// TIA Portal V17 program export: 0 tag tables, 0 data types, 40 data blocks, 87 code blocks (in call order from the OBs), 109 instance data blocks

DATA_BLOCK "General_DB"   // DB47
{ S7_Optimized_Access := 'TRUE' }
VERSION : 0.1
// stored: AutoNumber false, DBAccessibleFromOPCUA true, DBAccessibleFromWebserver true, IsOnlyStoredInLoadMemory false, IsRetainMemResEnabled false, IsWriteProtectedInAS false, MemoryReserve 100
   VAR
      Initial : Bool;
      "Reset HMI Prep" : Bool;
      "Reset HMI ST" : Bool;
      "Reset HMI Blend" : Bool;
      "Reset Scada" : Bool;
      Reset : Bool;
      Reset_Dose : Bool;
      Sim_Mode : Bool;   // 1 Simulation
      Sim_ON : Bool;
      Sim_OFF : Bool;
      Man_Initi : Bool;
      LDT_PLC : Date_And_Time;
      LDT_retval : Int;
      CIP_Line1_Open : Struct
         "CIP Tank_T01" : Bool;
         "CIP Line_T01" : Bool;
         "CIP Tank_T02" : Bool;
         "CIP Line_T02" : Bool;
         "CIP Tank_T03" : Bool;
         "CIP Line_T03" : Bool;
         "CIP Tank_T04" : Bool;
         "CIP Line_T04" : Bool;
         "CIP Tank_T05" : Bool;
         "CIP Line_T05" : Bool;
         "CIP Tank_T06" : Bool;
         "CIP Line_T06" : Bool;
         "CIP Tank_T07" : Bool;
         "CIP Line_T07" : Bool;
         "CIP Tank_T08" : Bool;
         "CIP Line_T08" : Bool;
         "CIP Tank_T09" : Bool;
         "CIP Line_T09" : Bool;
         "CIP Tank_T10" : Bool;
         "CIP Line_T10" : Bool;
         "CIP Tank_T11" : Bool;
         "CIP Line_T11" : Bool;
         "CIP Tank_T12" : Bool;
         "CIP Line_T12" : Bool;
         "CIP Tank_T13" : Bool;
         "CIP Line_T13" : Bool;
         CIP_Tank : Bool;
         CIP_Line : Bool;
      END_STRUCT;
      CIP_Line2_Open : Struct
         "CIP Tank_T1" : Bool;
         "CIP Line_T1" : Bool;
         "CIP Tank_T2" : Bool;
         "CIP Line_T2" : Bool;
         "CIP Tank_T3" : Bool;
         "CIP Line_T3" : Bool;
         "CIP Tank_T4" : Bool;
         "CIP Line_T4" : Bool;
         "CIP Tank_T5" : Bool;
         "CIP Line_T5" : Bool;
         "CIP Tank_T6" : Bool;
         "CIP Line_T6" : Bool;
         "CIP Tank_T7" : Bool;
         "CIP Line_T7" : Bool;
         "CIP Tank_T8" : Bool;
         "CIP Line_T8" : Bool;
         "CIP Tank_T9" : Bool;
         "CIP Line_T9" : Bool;
         "CIP Tank_T10" : Bool;
         "CIP Line_T10" : Bool;
         CIP_Tank : Bool;
         CIP_Line : Bool;
      END_STRUCT;
      "Bypass CIP Signal Storage" : Bool;
      "Bypass CIP Signal Homomixer" : Bool;
      "Testing FB Valve" : Struct
         Preparation : Bool;
         Homomixer : Bool;
         Blending : Bool;
         Storage : Bool;
      END_STRUCT;
      "Testing FB Motor" : Struct
         "MCC Blending" : Bool;
         "MCC Preparation" : Bool;
      END_STRUCT;
      "CIP Drain Time" : Struct
         BlendingCluster1 : TOF_TIME;
         BlendingCluster2 : TOF_TIME;
         "Preparation_02.20" : TOF_TIME;
         "Preparation_05.20" : TOF_TIME;
         Homomixer : TOF_TIME;
         "Storage_29.06" : TOF_TIME;
         "Storage_39.06" : TOF_TIME;
         HMI_Input : Struct
            BlendingCluster1 : Int := 60;
            BlendingCluster2 : Int := 60;
            "Preparation_02.20" : Int := 60;
            "Preparation_05.20" : Int := 60;
            Homomixer : Int := 60;
            "Storage_29.06" : Int := 60;
            "Storage_39.06" : Int := 60;
         END_STRUCT;
         Actual : Struct
            BlendingCluster1 : DInt;
            BlendingCluster2 : DInt;
            "Preparation_02.20" : DInt;
            "Preparation_05.20" : DInt;
            Homomixer : DInt;
            "Storage_29.06" : DInt;
            "Storage_39.06" : DInt;
         END_STRUCT;
      END_STRUCT;
   END_VAR
BEGIN
   "CIP Drain Time".BlendingCluster1.PT := T#1m;
   "CIP Drain Time".BlendingCluster2.PT := T#1m;
   "CIP Drain Time"."Preparation_02.20".PT := T#1m;
   "CIP Drain Time"."Preparation_05.20".PT := T#1m;
   "CIP Drain Time".Homomixer.PT := T#1m;
   "CIP Drain Time"."Storage_29.06".PT := T#1m;
   "CIP Drain Time"."Storage_39.06".PT := T#1m;
END_DATA_BLOCK

DATA_BLOCK "General_Blend"   // DB33
{ S7_Optimized_Access := 'TRUE' }
VERSION : 0.1
// stored: AutoNumber true, DBAccessibleFromOPCUA true, DBAccessibleFromWebserver true, IsOnlyStoredInLoadMemory false, IsRetainMemResEnabled false, IsWriteProtectedInAS false, MemoryReserve 100
   VAR
      Drain_ON_OFF_THE1 : Bool;
      Drain_ON_OFF_THE2 : Bool;
      Blend_Cluster1 : Struct
         CIP_Line1 : Struct
            "CIP Enable" : Bool;
            "CIP Request" : Bool;
            V_Cmd : Bool;
            P_Cmd : Bool;
            P_SP : Real;
         END_STRUCT;
         CIP_Line2 : Struct
            "CIP Enable" : Bool;
            "CIP Request" : Bool;
            V_Cmd : Bool;
            P_Cmd : Bool;
            P_SP : Real;
         END_STRUCT;
         CIP_Line3 : Struct
            "CIP Enable" : Bool;
            "CIP Request" : Bool;
            V_Cmd : Bool;
            P_Cmd : Bool;
            P_SP : Real;
         END_STRUCT;
         ptrig : Bool;
      END_STRUCT;
      Blend_Cluster2 : Struct
         CIP_Line1 : Struct
            "CIP Enable" : Bool;
            "CIP Request" : Bool;
            V_Cmd : Bool;
            P_Cmd : Bool;
            P_SP : Real;
         END_STRUCT;
         CIP_Line2 : Struct
            "CIP Enable" : Bool;
            "CIP Request" : Bool;
            V_Cmd : Bool;
            P_Cmd : Bool;
            P_SP : Real;
         END_STRUCT;
         CIP_Line3 : Struct
            "CIP Enable" : Bool;
            "CIP Request" : Bool;
            V_Cmd : Bool;
            P_Cmd : Bool;
            P_SP : Real;
         END_STRUCT;
         ptrig : Bool;
      END_STRUCT;
      CIP_Bypass : Bool;
      "THE-4" : Struct
         "Timer" : TON_TIME;
         MSec { S7_SetPoint := 'True'} : DInt;
         Sec : DInt := 10;
         Act : DInt;
      END_STRUCT;
      "THE-5" : Struct
         "Timer" : TON_TIME;
         MSec { S7_SetPoint := 'True'} : DInt;
         Sec : DInt := 10;
         Act : DInt;
      END_STRUCT;
      Sugar : Struct
         "In Process" : Struct
            "T-20" : Bool;
            "T-21" : Bool;
            "T-30" : Bool;
            "T-31" : Bool;
            "T-40" : Bool;
            "T-41" : Bool;
         END_STRUCT;
      END_STRUCT;
   END_VAR
BEGIN
END_DATA_BLOCK

DATA_BLOCK "Gen_Storage"   // DB15
{ S7_Optimized_Access := 'TRUE' }
VERSION : 0.1
// stored: AutoNumber false, DBAccessibleFromOPCUA true, DBAccessibleFromWebserver true, IsOnlyStoredInLoadMemory false, IsRetainMemResEnabled false, IsWriteProtectedInAS false, MemoryReserve 100
   VAR
      "Timer" : Struct
         Off_DrainIn_23 : TOF_TIME;
         Off_DrainIn_24_1 { S7_SetPoint := 'True'} : TOF_TIME;
         Off_DrainIn_24_2 { S7_SetPoint := 'True'} : TOF_TIME;
         Off_DrainIn_33 { S7_SetPoint := 'True'} : TOF_TIME;
         Off_DrainIn_34 { S7_SetPoint := 'True'} : TOF_TIME;
         Off_DrainIn_35 { S7_SetPoint := 'True'} : TOF_TIME;
         Off_DrainIn_79_1 { S7_SetPoint := 'True'} : TOF_TIME;
         Off_DrainIn_79_2 { S7_SetPoint := 'True'} : TOF_TIME;
         Off_DrainIn_79_3 { S7_SetPoint := 'True'} : TOF_TIME;
         Off_DrainIn_81 { S7_SetPoint := 'True'} : TOF_TIME;
         Off_DrainIn_84 { S7_SetPoint := 'True'} : TOF_TIME;
         Off_DrainIn_85 { S7_SetPoint := 'True'} : TOF_TIME;
      END_STRUCT;
      "THE4 CIP" : Struct
         "CIP Enable" : Bool;
         "CIP Request" : Bool;
         "CIP Line OK" : Bool;
         "CIP on Prog" : Bool;
         V_CIP_Cmd : Bool;
         p_trig : Bool;
      END_STRUCT;
      "THE5 CIP" : Struct
         "CIP Enable" : Bool;
         "CIP Request" : Bool;
         "CIP Line OK" : Bool;
         "CIP on Prog" : Bool;
         V_CIP_Cmd : Bool;
         p_trig : Bool;
      END_STRUCT;
   END_VAR
BEGIN
   "Timer".Off_DrainIn_23.PT := T#3s;
   "Timer".Off_DrainIn_24_1.PT := T#3s;
   "Timer".Off_DrainIn_33.PT := T#3s;
   "Timer".Off_DrainIn_34.PT := T#3s;
   "Timer".Off_DrainIn_35.PT := T#3s;
   "Timer".Off_DrainIn_79_1.PT := T#3s;
   "Timer".Off_DrainIn_81.PT := T#3s;
   "Timer".Off_DrainIn_84.PT := T#3s;
   "Timer".Off_DrainIn_85.PT := T#3s;
END_DATA_BLOCK

DATA_BLOCK "General Preparation"   // DB59
{ S7_Optimized_Access := 'TRUE' }
VERSION : 0.1
// stored: AutoNumber true, DBAccessibleFromOPCUA true, DBAccessibleFromWebserver true, IsOnlyStoredInLoadMemory false, IsRetainMemResEnabled false, IsWriteProtectedInAS false, MemoryReserve 100
   VAR
      "Header 1" : Struct
         "CIP Enable" : Bool;
         "CIP Request" : Bool;
         "CIP Line OK" : Bool;
         "CIP on Prog" : Bool;
         V_CIP_Cmd : Bool;
         p_trig : Bool;
      END_STRUCT;
      "Header 2" : Struct
         "CIP Enable" : Bool;
         "CIP Request" : Bool;
         "CIP Line OK" : Bool;
         "CIP on Prog" : Bool;
         V_CIP_Cmd : Bool;
         p_trig : Bool;
      END_STRUCT;
      "Blend OSA" : Struct
         "CIP Enable_T-06 Cmd" : Bool;
         "CIP Enable_T-07 Cmd" : Bool;
         "CIP Enable_T-08 Cmd" : Bool;
         "CIP Request" : Bool;
         "CIP on Prog" : Bool;
         "CIP EN T-06" : Bool;
         "CIP EN T-07" : Bool;
         "CIP EN T-08" : Bool;
      END_STRUCT;
      "Tipper 1" : Struct
         "CIP Enable Cmd" : Bool;
         "CIP Request" : Bool;
         "CIP on Prog" : Bool;
         "CIP EN" : Bool;
      END_STRUCT;
      "Tipper 2" : Struct
         "CIP Enable_T-03 Cmd" : Bool;
         "CIP Enable_T-04 Cmd" : Bool;
         "CIP Request" : Bool;
         "CIP on Prog" : Bool;
         "CIP EN T-03" : Bool;
         "CIP EN T-04" : Bool;
      END_STRUCT;
      CIP_Bypass : Bool;
      Reset_Totalizer : Struct
         "FT_T-51" : Bool;
         "FT_T-02" : Bool;
         "FT_T-3" : Bool;
         "FT_T-4" : Bool;
         "FT_T-5" : Bool;
         "FT_T-6" : Bool;
         "FT_T-7" : Bool;
         "FT_T-8" : Bool;
         "FT_T-9" : Bool;
         "FT_T-10" : Bool;
      END_STRUCT;
      CV_Value_Manual : Real;
   END_VAR
   VAR RETAIN
      Tank_Name : Struct
         ChiliAwetan1 : String := 'Chili Awetan 1';
         ChiliAwetan2 : String := 'Chili Awetan 2';
         ChiliAwetan3 : String := 'Chili Awetan 3';
         Tomato : String := 'Tomato';
         ChiliFresh1 : String := 'Chili Fresh 1';
         ChiliFresh2 : String := 'Chili Fresh 2';
         ChiliFresh3 : String := 'Chili Fresh 3';
         Garlic : String := 'Garlic';
         Vinegar : String := 'Vinegar';
         HotWater : String := 'Hot Water';
         free11 : String;
      END_STRUCT;
   END_VAR
BEGIN
END_DATA_BLOCK

DATA_BLOCK "General Buffer"   // DB63
{ S7_Optimized_Access := 'TRUE' }
VERSION : 0.1
// stored: AutoNumber true, DBAccessibleFromOPCUA true, DBAccessibleFromWebserver true, IsOnlyStoredInLoadMemory false, IsRetainMemResEnabled false, IsWriteProtectedInAS false, MemoryReserve 100
   VAR
      "CIP Enable" : Struct
         Cluster1_Line3 : Bool;
         Cluster2_Line1 : Bool;
         Cluster2_Line2 : Bool;
         Cluster2_Line3 : Bool;
      END_STRUCT;
      "CIP Line Open" : Struct
         Cluster1_Line3 : Bool;
         Cluster2_Line1 : Bool;
         Cluster2_Line2 : Bool;
         Cluster2_Line3 : Bool;
      END_STRUCT;
   END_VAR
BEGIN
END_DATA_BLOCK

DATA_BLOCK "CIP_CIP_to_Sto"   // DB190
{ S7_Optimized_Access := 'FALSE' }
VERSION : 0.1
// stored: AutoNumber false, DBAccessibleFromOPCUA true, DBAccessibleFromWebserver true, IsOnlyStoredInLoadMemory false, IsWriteProtectedInAS false
   VAR
      HeatBeat : Bool;
      CIP_Ready : Bool;   // Cip Kitchen Ready
      CIP_Inprogress : Bool;   // Reqquest approved
      CIP_Complete : Bool;
      Valve_Line_Return_Open : Bool;
      Spare : Bool;
      Spare_1 : Bool;
      Spare_2 : Bool;
      Spare_3 : Bool;
      Spare_4 : Bool;
      Spare_5 : Bool;
      Spare_6 : Bool;
      Spare_7 : Bool;
      Spare_8 : Bool;
      Spare_9 : Bool;
      Spare_10 : Bool;
      Data_Real : Real;
      Data_Real_1 : Real;
      Data_Real_2 : Real;
      Data_Real_3 : Real;
      Data_Real_4 : Real;
      Data_Real_5 : Real;
      Data_Real_6 : Real;
      Data_Real_7 : Real;
   END_VAR
BEGIN
END_DATA_BLOCK

DATA_BLOCK "CIP_Sto_to_CIP"   // DB191
{ S7_Optimized_Access := 'FALSE' }
VERSION : 0.1
// stored: AutoNumber false, DBAccessibleFromOPCUA true, DBAccessibleFromWebserver true, IsOnlyStoredInLoadMemory false, IsWriteProtectedInAS false
   VAR
      HeatBeat : Bool;
      CIP_Request : Bool;   // Cip Kitchen Ready
      ReturnPump_ON : Bool;   // Reqquest approved
      CIP_Complete : Bool;
      Valve_Line_Supply_Open : Bool;
      Spare : Bool;
      Spare_1 : Bool;
      Spare_2 : Bool;
      Spare_3 : Bool;
      Spare_4 : Bool;
      Spare_5 : Bool;
      Spare_6 : Bool;
      Spare_7 : Bool;
      Spare_8 : Bool;
      Spare_9 : Bool;
      Spare_10 : Bool;
      Data_Real : Real;
      Data_Real_1 : Real;
      Data_Real_2 : Real;
      Data_Real_3 : Real;
      Data_Real_4 : Real;
      Data_Real_5 : Real;
      Data_Real_6 : Real;
      Data_Real_7 : Real;
   END_VAR
BEGIN
END_DATA_BLOCK

DATA_BLOCK "CommSett_DB"   // DB10
{ S7_Optimized_Access := 'TRUE' }
VERSION : 0.1
// stored: AutoNumber false, DBAccessibleFromOPCUA true, DBAccessibleFromWebserver true, IsOnlyStoredInLoadMemory false, IsRetainMemResEnabled false, IsWriteProtectedInAS false, MemoryReserve 100
   VAR
      THE1_put : "typePut";
      THE1_get { S7_SetPoint := 'True'} : "typeGet";
      THE1_diagnostic { S7_SetPoint := 'True'} : "typeDiagnostic";
      THE2_put : "typePut";
      THE2_get { S7_SetPoint := 'True'} : "typeGet";
      THE2_diagnostic { S7_SetPoint := 'True'} : "typeDiagnostic";
      THE1_Comm_Error { S7_SetPoint := 'True'} : Bool;
      THE2_Comm_Error : Bool;
      THE1_Comm : Array[0..10] of Byte;
      THE2_Comm : Array[0..10] of Byte;
      CIP_put : "typePut";
      CIP_get { S7_SetPoint := 'True'} : "typeGet";
      CIP_diagnostic { S7_SetPoint := 'True'} : "typeDiagnostic";
      CIP_Comm_Error { S7_SetPoint := 'True'} : Bool;
      CIP_Comm : Array[0..10] of Byte;
   END_VAR
BEGIN
   THE1_put.connectionId := 16#100;
   THE1_get.connectionId := 16#100;
   THE2_put.connectionId := 16#101;
   THE2_get.connectionId := 16#101;
   CIP_put.connectionId := 16#102;
   CIP_get.connectionId := 16#102;
END_DATA_BLOCK

DATA_BLOCK "Data_block_1"   // DB196
{ S7_Optimized_Access := 'FALSE'; DB_Accessible_From_OPC_UA := 'FALSE' }
VERSION : 0.1
// stored: AutoNumber false, DBAccessibleFromOPCUA false, DBAccessibleFromWebserver false, IsOnlyStoredInLoadMemory false, IsWriteProtectedInAS false
   VAR
      FromTHE4 : Array[0..50] of Byte;
   END_VAR
BEGIN
END_DATA_BLOCK

DATA_BLOCK "THE1_From_BT_To_Mixing"   // DB194
{ S7_Optimized_Access := 'FALSE' }
VERSION : 0.1
// stored: AutoNumber false, DBAccessibleFromOPCUA true, DBAccessibleFromWebserver true, IsOnlyStoredInLoadMemory false, IsWriteProtectedInAS false
   VAR RETAIN
      HeartBeat : Bool := TRUE;
      CIPEnable : Bool;
      LineProd_Open : Bool;
      LineCIP_Open : Bool;
      _free_4 : Bool;
      _free_5 : Bool;
      _free_6 : Bool;
      _free_7 : Bool;
      ProductRequest : Bool;
      _free_09 : Bool;
      _free_10 : Bool;
      _free_11 : Bool;
      _free_12 : Bool;
      _free_13 : Bool;
      _free_14 : Bool;
      _free_15 : Bool;
      _free_real2 : Real;
      _free_real6 : Real := 20000.0;
      _free_real10 : Real;
      _free_real14 : Real;
      _free_real18 : Real;
      _free_real22 : Real;
      _free_real26 : Real;
      _free_real30 : Real;
      FromTHE1Byte1 : Byte;
      FromTHE1Byte2 : Byte;
      FromTHE1Byte3 : Byte;
      FromTHE1Byte4 : Byte;
   END_VAR
BEGIN
END_DATA_BLOCK

DATA_BLOCK "THE1_From_Mixing_To_BT"   // DB195
{ S7_Optimized_Access := 'FALSE' }
VERSION : 0.1
// stored: AutoNumber false, DBAccessibleFromOPCUA true, DBAccessibleFromWebserver true, IsOnlyStoredInLoadMemory false, IsWriteProtectedInAS false
   VAR RETAIN
      HeartBeat : Bool;
      CIPRequest : Bool;
      MixProofFlip : Bool;
      Drain_valve : Bool;
      _free_4 : Bool;
      _free_5 : Bool;
      _free_6 : Bool;
      _free_7 : Bool;
      ProductAvailable : Bool;
      ProductTransferInProgress : Bool;
      _free_10 : Bool;
      _free_11 : Bool;
      _free_12 : Bool;
      _free_13 : Bool;
      _free_14 : Bool;
      _free_15 : Bool;
      _free_real2 : Real := 52.25618;
      _free_real6 : Real := 93.70135;
      _free_real10 : Real := 95.52147;
      _free_real14 : Real := 90.2006;
      _free_real18 : Real;
      _free_real22 : Real;
      _free_real26 : Real;
      _free_real30 : Real;
      ForTHE1_Byte1 : Byte;
      ForTHE1_Byte2 : Byte;
      ForTHE1_Byte3 : Byte;
      ForTHE1_Byte4 : Byte;
   END_VAR
BEGIN
END_DATA_BLOCK

DATA_BLOCK "THE2_From_BT_To_Mixing"   // DB198
{ S7_Optimized_Access := 'FALSE' }
VERSION : 0.1
// stored: AutoNumber false, DBAccessibleFromOPCUA true, DBAccessibleFromWebserver true, IsOnlyStoredInLoadMemory false, IsWriteProtectedInAS false
   VAR RETAIN
      HeartBeat : Bool := TRUE;
      CIPEnable : Bool;
      LineProd_Open : Bool;
      LineCIP_Open : Bool;
      _free_4 : Bool;
      _free_5 : Bool;
      _free_6 : Bool;
      _free_7 : Bool;
      ProductRequest : Bool;
      _free_09 : Bool;
      _free_10 : Bool;
      _free_11 : Bool;
      _free_12 : Bool;
      _free_13 : Bool;
      _free_14 : Bool;
      _free_15 : Bool;
      _free_real2 : Real;
      _free_real6 : Real := 20000.0;
      _free_real10 : Real;
      _free_real14 : Real;
      _free_real18 : Real;
      _free_real22 : Real;
      _free_real26 : Real;
      _free_real30 : Real;
      FromTHE2Byte1 : Byte;
      FromTHE2Byte2 : Byte;
      FromTHE2Byte3 : Byte;
      FromTHE2Byte4 : Byte;
   END_VAR
BEGIN
END_DATA_BLOCK

DATA_BLOCK "THE2_From_Mixing_To_BT"   // DB199
{ S7_Optimized_Access := 'FALSE' }
VERSION : 0.1
// stored: AutoNumber false, DBAccessibleFromOPCUA true, DBAccessibleFromWebserver true, IsOnlyStoredInLoadMemory false, IsWriteProtectedInAS false
   VAR RETAIN
      HeartBeat : Bool;
      CIPRequest : Bool;
      MixProofFlip : Bool;
      Drain_valve : Bool;
      _free_4 : Bool;
      _free_5 : Bool;
      _free_6 : Bool;
      _free_7 : Bool;
      ProductAvailable : Bool;
      ProductTransferInProgress : Bool;
      _free_10 : Bool;
      _free_11 : Bool;
      _free_12 : Bool;
      _free_13 : Bool;
      _free_14 : Bool;
      _free_15 : Bool;
      _free_real2 : Real := 52.25618;
      _free_real6 : Real := 93.70135;
      _free_real10 : Real := 95.52147;
      _free_real14 : Real := 90.2006;
      _free_real18 : Real;
      _free_real22 : Real;
      _free_real26 : Real;
      _free_real30 : Real;
      ForTHE2_Byte1 : Byte;
      ForTHE2_Byte2 : Byte;
      ForTHE2_Byte3 : Byte;
      ForTHE2_Byte4 : Byte;
   END_VAR
BEGIN
END_DATA_BLOCK

DATA_BLOCK "MB to Osa"   // DB265
{ S7_Optimized_Access := 'FALSE' }
VERSION : 0.1
// stored: AutoNumber false, DBAccessibleFromOPCUA true, DBAccessibleFromWebserver true, IsOnlyStoredInLoadMemory false, IsWriteProtectedInAS false
   VAR
      HeartBeat : Bool;   // Clock 1Hz
      ChiliFresh1_Prod_Req : Bool;
      ChiliFresh2_Prod_Req : Bool;
      ChiliFresh3_Prod_Req : Bool;
      ChiliFresh1_Line_OK : Bool;
      ChiliFresh2_Line_OK : Bool;
      ChiliFresh3_Line_OK : Bool;
      ChiliFresh1_CIP_Enable : Bool;
      ChiliFresh2_CIP_Enable : Bool;
      ChiliFresh3_CIP_Enable : Bool;
      freeBool11 : Bool;
      freeBool12 : Bool;
      freeBool13 : Bool;
      freeBool14 : Bool;
      freeBool15 : Bool;
      freeBool16 : Bool;
      freeBool17 : Bool;
   END_VAR
BEGIN
END_DATA_BLOCK

DATA_BLOCK "Osa to MB"   // DB264
{ S7_Optimized_Access := 'FALSE' }
VERSION : 0.1
// stored: AutoNumber false, DBAccessibleFromOPCUA true, DBAccessibleFromWebserver true, IsOnlyStoredInLoadMemory false, IsWriteProtectedInAS false
   VAR
      HeartBeat : Bool;   // Clock 1hz
      Product_Ready : Bool;
      Product_LineOpen : Bool;
      Product_SupplyON : Bool;
      Product_Transfer_Complete : Bool;
      freeBool5 : Bool;
      freeBool6 : Bool;
      freeBool7 : Bool;
      freeBool8 : Bool;
      freeBool9 : Bool;
      freeBool10 : Bool;
      freeBool11 : Bool;
      freeBool12 : Bool;
      freeBool13 : Bool;
      freeBool14 : Bool;
      freeBool15 : Bool;
      freeBool16 : Bool;
      freeBool17 : Bool;
      freeBool18 : Bool;
      freeBool19 : Bool;
      freeBool20 : Bool;
      freeBool21 : Bool;
      freeBool22 : Bool;
      freeBool23 : Bool;
   END_VAR
BEGIN
END_DATA_BLOCK

DATA_BLOCK "CIP_to_Mix"   // DB220
{ S7_Optimized_Access := 'FALSE' }
VERSION : 0.1
// stored: AutoNumber false, DBAccessibleFromOPCUA true, DBAccessibleFromWebserver true, IsOnlyStoredInLoadMemory false, IsWriteProtectedInAS false
   VAR
      HeartBeat : Bool := TRUE;
      CIP_RequestOK : Struct
         Header : Struct
            Header_CIP_RequestOK : Bool;
         END_STRUCT;
         "Chili Awetan" : Struct
            "T-02.00_CIP_RequestOK" : Bool;
            "T-03.00_CIP_RequestOK" : Bool;
            "T-04.00_CIP_RequestOK" : Bool;
         END_STRUCT;
         Tomato : Struct
            "T-05.00_CIP_RequestOK" : Bool;
         END_STRUCT;
         ChiliFresh : Struct
            "T-06.00_CIP_RequestOK" : Bool;
            "T-07.00_CIP_RequestOK" : Bool;
            "T-08.00_CIP_RequestOK" : Bool;
         END_STRUCT;
         Garlic : Struct
            "T-09.00_CIP_RequestOK" : Bool;
         END_STRUCT;
         Vinegar : Struct
            "T-10.00_CIP_RequestOK" : Bool;
         END_STRUCT;
         Homomixer : Struct
            "T-12.00_CIP_RequestOK" : Bool;
            "T-13.00_CIP_RequestOK" : Bool;
            "T-14.00_CIP_RequestOK" : Bool;
         END_STRUCT;
         "Blending Cluster 1" : Struct
            "T-20.00_CIP_RequestOK" : Bool;
            "T-21.00_CIP_RequestOK" : Bool;
            "T-30.00_CIP_RequestOK" : Bool;
            Blending_Cluster1_LineProduct_RequestOK : Bool;
            Free_CIP_RequestOK_1 : Bool;
            Free_CIP_RequestOK_2 : Bool;
         END_STRUCT;
         "Blending Cluster 2" : Struct
            "T-31.00_CIP_RequestOK" : Bool;
            "T-40.00_CIP_RequestOK" : Bool;
            "T-41.00_CIP_RequestOK" : Bool;
            Blending_Cluster2_LineProduct_RequestOK : Bool;
            Free_CIP_RequestOK_1 : Bool;
            Free_CIP_RequestOK_2 : Bool;
         END_STRUCT;
         "Rework Cluster 1" : Struct
            "T-22.00_CIP_RequestOK" : Bool;
         END_STRUCT;
         "Rework Cluster 2" : Struct
            "T-32.00_CIP_RequestOK" : Bool;
         END_STRUCT;
         "Buffer Cluster 1" : Struct
            "T-61.00_CIP_RequestOK" : Bool;
            "T-62.00_CIP_RequestOK" : Bool;
            "T61&T62_CIP_LineToPasteur_RequestOK" : Bool;
            "T-63.00_CIP_RequestOK" : Bool;
            "T-64.00_CIP_RequestOK" : Bool;
            "T63&T64_CIP_LineToPasteur_RequestOK" : Bool;
         END_STRUCT;
         "Buffer Cluster 2" : Struct
            "T-65.00_CIP_RequestOK" : Bool;
            "T-66.00_CIP_RequestOK" : Bool;
            "T65&T66_CIP_LineToPasteur_RequestOK" : Bool;
            "T-67.00_CIP_RequestOK" : Bool;
            "T-68.00_CIP_RequestOK" : Bool;
            "T67&T68_CIP_LineToPasteur_RequestOK" : Bool;
         END_STRUCT;
         "Storage THE 4" : Struct
            "T-23.00_CIP_RequestOK" : Bool;
            "T-24.00_CIP_RequestOK" : Bool;
            THE4_LineProduct_CIP_RequestOK : Bool;
         END_STRUCT;
         "Storage THE 5" : Struct
            "T-33.00_CIP_Tank_RequestOK" : Bool;
            "T-34.00_CIP_Tank_RequestOK" : Bool;
            "T33&T34_CIP_Line_RequestOK" : Bool;
            "T-35.00_CIP_Tank_RequestOK" : Bool;
            THE5_LineProduct_CIP_RequestOK : Bool;
         END_STRUCT;
         "T-79.00_CIP_RequestOK" : Bool;
         "T-81.00_CIP_RequestOK" : Bool;
         "T-84.00_CIP_RequestOK" : Bool;
         "T-85.00_CIP_RequestOK" : Bool;
         JBT_THE4_RequestOK : Bool;   // Open AV-22.11
         JBT_THE5_RequestOK : Bool;   // Open AV-22.11
         Aseptic_Pharmac_RequestOK : Bool;   // Open AV-39.06
         Free_CIP_RequestOK_8 : Bool;
         Free_CIP_RequestOK_9 : Bool;
         Free_CIP_RequestOK_10 : Bool;
         Free_CIP_RequestOK_11 : Bool;
         Free_CIP_RequestOK_12 : Bool;
         Free_CIP_RequestOK_13 : Bool;
         Free_CIP_RequestOK_14 : Bool;
         Free_CIP_RequestOK_15 : Bool;
         Free_CIP_RequestOK_16 : Bool;
         Osa_CIP_RequestOK : Bool;
         Free_CIP_RequestOK_18 : Bool;
         Free_CIP_RequestOK_19 : Bool;
         Free_CIP_RequestOK_20 : Bool;
         Free_CIP_RequestOK_21 : Bool;
         Free_CIP_RequestOK_22 : Bool;
         Free_CIP_RequestOK_23 : Bool;
         Free_CIP_RequestOK_24 : Bool;
      END_STRUCT;
      CIP_InProgress : Struct
         Header : Struct
            Header_CIP_InProgress : Bool;
         END_STRUCT;
         "Chili Awetan" : Struct
            "T-02.00_CIP_InProgress" : Bool;
            "T-03.00_CIP_InProgress" : Bool;
            "T-04.00_CIP_InProgress" : Bool;
         END_STRUCT;
         Tomato : Struct
            "T-05.00_CIP_InProgress" : Bool;
         END_STRUCT;
         ChiliFresh : Struct
            "T-06.00_CIP_InProgress" : Bool;
            "T-07.00_CIP_InProgress" : Bool;
            "T-08.00_CIP_InProgress" : Bool;
         END_STRUCT;
         Garlic : Struct
            "T-09.00_CIP_InProgress" : Bool;
         END_STRUCT;
         Vinegar : Struct
            "T-10.00_CIP_InProgress" : Bool;
         END_STRUCT;
         Homomixer : Struct
            "T-12.00_CIP_InProgress" : Bool;
            "T-13.00_CIP_InProgress" : Bool;
            "T-14.00_CIP_InProgress" : Bool;
         END_STRUCT;
         "Blending Cluster 1" : Struct
            "T-20.00_CIP_InProgress" : Bool;
            "T-21.00_CIP_InProgress" : Bool;
            "T-30.00_CIP_InProgress" : Bool;
            Blending_Cluster1_LineProduct_InProgress : Bool;
            Free_CIP_InProgress_1 : Bool;
            Free_CIP_InProgress_2 : Bool;
         END_STRUCT;
         "Blending Cluster 2" : Struct
            "T-31.00_CIP_InProgress" : Bool;
            "T-40.00_CIP_InProgress" : Bool;
            "T-41.00_CIP_InProgress" : Bool;
            Blending_Cluster2_LineProduct_InProgress : Bool;
            Free_CIP_InProgress_1 : Bool;
            Free_CIP_InProgress_2 : Bool;
         END_STRUCT;
         "Rework Cluster 1" : Struct
            "T-22.00_CIP_InProgress" : Bool;
         END_STRUCT;
         "Rework Cluster 2" : Struct
            "T-32.00_CIP_InProgress" : Bool;
         END_STRUCT;
         "Buffer Cluster 1" : Struct
            "T-61.00_CIP_InProgress" : Bool;
            "T-62.00_CIP_InProgress" : Bool;
            "T61&T62_CIP_LineToPasteur_InProgress" : Bool;
            "T-63.00_CIP_InProgress" : Bool;
            "T-64.00_CIP_InProgress" : Bool;
            "T63&T64_CIP_LineToPasteur_InProgress" : Bool;
         END_STRUCT;
         "Buffer Cluster 2" : Struct
            "T-65.00_CIP_InProgress" : Bool;
            "T-66.00_CIP_InProgress" : Bool;
            "T65&T66_CIP_LineToPasteur_InProgress" : Bool;
            "T-67.00_CIP_InProgress" : Bool;
            "T-68.00_CIP_InProgress" : Bool;
            "T67&T68_CIP_LineToPasteur_InProgress" : Bool;
         END_STRUCT;
         "Storage THE 4" : Struct
            "T-23.00_CIP_InProgress" : Bool;
            "T-24.00_CIP_InProgress" : Bool;
            THE4_LineProduct_CIP_InProgress : Bool;
         END_STRUCT;
         "Storage THE 5" : Struct
            "T-33.00_CIP_Tank_InProgress" : Bool;
            "T-34.00_CIP_Tank_InProgress" : Bool;
            "T33&T34_CIP_Line_InProgress" : Bool;
            "T-35.00_CIP_Tank_InProgress" : Bool;
            THE5_LineProduct_CIP_InProgress : Bool;
         END_STRUCT;
         "T-79.00_CIP_InProgress" : Bool;
         "T-81.00_CIP_InProgress" : Bool;
         "T-84.00_CIP_InProgress" : Bool;
         "T-85.00_CIP_InProgress" : Bool;
         Free_CIP_InProgress_5 : Bool;
         Free_CIP_InProgress_6 : Bool;
         Free_CIP_InProgress_7 : Bool;
         Free_CIP_InProgress_8 : Bool;
         Free_CIP_InProgress_9 : Bool;
         Free_CIP_InProgress_10 : Bool;
         Free_CIP_InProgress_11 : Bool;
         Free_CIP_InProgress_12 : Bool;
         Free_CIP_InProgress_13 : Bool;
         Free_CIP_InProgress_14 : Bool;
         Free_CIP_InProgress_15 : Bool;
         Free_CIP_InProgress_16 : Bool;
         Osa_CIP_InProgress : Bool;
         Free_CIP_InProgress_18 : Bool;
         Free_CIP_InProgress_19 : Bool;
         Free_CIP_InProgress_20 : Bool;
         Free_CIP_InProgress_21 : Bool;
         Free_CIP_InProgress_22 : Bool;
         Free_CIP_InProgress_23 : Bool;
         Free_CIP_InProgress_24 : Bool;
      END_STRUCT;
      CIP_Supply_On : Struct
         Header : Struct
            Header_CIP_Supply_ON : Bool;
         END_STRUCT;
         "Chili Awetan" : Struct
            "T-02.00_CIP_Supply_ON" : Bool;
            "T-03.00_CIP_Supply_ON" : Bool;
            "T-04.00_CIP_Supply_ON" : Bool;
         END_STRUCT;
         Tomato : Struct
            "T-05.00_CIP_Supply_ON" : Bool;
         END_STRUCT;
         ChiliFresh : Struct
            "T-06.00_CIP_Supply_ON" : Bool;
            "T-07.00_CIP_Supply_ON" : Bool;
            "T-08.00_CIP_Supply_ON" : Bool;
         END_STRUCT;
         Garlic : Struct
            "T-09.00_CIP_Supply_ON" : Bool;
         END_STRUCT;
         Vinegar : Struct
            "T-10.00_CIP_Supply_ON" : Bool;
         END_STRUCT;
         Homomixer : Struct
            "T-12.00_CIP_Supply_ON" : Bool;
            "T-13.00_CIP_Supply_ON" : Bool;
            "T-14.00_CIP_Supply_ON" : Bool;
         END_STRUCT;
         "Blending Cluster 1" : Struct
            "T-20.00_CIP_Supply_ON" : Bool;
            "T-21.00_CIP_Supply_ON" : Bool;
            "T-30.00_CIP_Supply_ON" : Bool;
            Blending_Cluster1_LineProduct_Supply_ON : Bool;
            Free_CIP_Supply_ON_1 : Bool;
            Free_CIP_Supply_ON_2 : Bool;
         END_STRUCT;
         "Blending Cluster 2" : Struct
            "T-31.00_CIP_Supply_ON" : Bool;
            "T-40.00_CIP_Supply_ON" : Bool;
            "T-41.00_CIP_Supply_ON" : Bool;
            Blending_Cluster2_LineProduct_Supply_ON : Bool;
            Free_CIP_Supply_ON_1 : Bool;
            Free_CIP_Supply_ON_2 : Bool;
         END_STRUCT;
         "Rework Cluster 1" : Struct
            "T-22.00_CIP_Supply_ON" : Bool;
         END_STRUCT;
         "Rework Cluster 2" : Struct
            "T-32.00_CIP_Supply_ON" : Bool;
         END_STRUCT;
         "Buffer Cluster 1" : Struct
            "T-61.00_CIP_Supply_ON" : Bool;
            "T-62.00_CIP_Supply_ON" : Bool;
            "T61&T62_CIP_LineToPasteur_Supply_ON" : Bool;
            "T-63.00_CIP_Supply_ON" : Bool;
            "T-64.00_CIP_Supply_ON" : Bool;
            "T63&T64_CIP_LineToPasteur_Supply_ON" : Bool;
         END_STRUCT;
         "Buffer Cluster 2" : Struct
            "T-65.00_CIP_Supply_ON" : Bool;
            "T-66.00_CIP_Supply_ON" : Bool;
            "T65&T66_CIP_LineToPasteur_Supply_ON" : Bool;
            "T-67.00_CIP_Supply_ON" : Bool;
            "T-68.00_CIP_Supply_ON" : Bool;
            "T67&T68_CIP_LineToPasteur_Supply_ON" : Bool;
         END_STRUCT;
         "Storage THE 4" : Struct
            "T-23.00_CIP_Supply_ON" : Bool;
            "T-24.00_CIP_Supply_ON" : Bool;
            THE4_LineProduct_CIP_Supply_ON : Bool;
         END_STRUCT;
         "Storage THE 5" : Struct
            "T-33.00_CIP_Tank_Supply_ON" : Bool;
            "T-34.00_CIP_Tank_Supply_ON" : Bool;
            "T33&T34_CIP_Line_Supply_ON" : Bool;
            "T-35.00_CIP_Tank_Supply_ON" : Bool;
            THE5_LineProduct_CIP_Supply_ON : Bool;
         END_STRUCT;
         "T-79.00_CIP_Supply_ON" : Bool;
         "T-81.00_CIP_Supply_ON" : Bool;
         "T-84.00_CIP_Supply_ON" : Bool;
         "T-85.00_CIP_Supply_ON" : Bool;
         Free_CIP_Supply_ON_5 : Bool;
         Free_CIP_Supply_ON_6 : Bool;
         Free_CIP_Supply_ON_7 : Bool;
         Free_CIP_Supply_ON_8 : Bool;
         Free_CIP_Supply_ON_9 : Bool;
         Free_CIP_Supply_ON_10 : Bool;
         Free_CIP_Supply_ON_11 : Bool;
         Free_CIP_Supply_ON_12 : Bool;
         Free_CIP_Supply_ON_13 : Bool;
         Free_CIP_Supply_ON_14 : Bool;
         Free_CIP_Supply_ON_15 : Bool;
         Free_CIP_Supply_ON_16 : Bool;
         Osa_CIP_Supply_ON : Bool;
         Free_CIP_Supply_ON_18 : Bool;
         Free_CIP_Supply_ON_19 : Bool;
         Free_CIP_Supply_ON_20 : Bool;
         Free_CIP_Supply_ON_21 : Bool;
         Free_CIP_Supply_ON_22 : Bool;
         Free_CIP_Supply_ON_23 : Bool;
         Free_CIP_Supply_ON_24 : Bool;
      END_STRUCT;
      CIP_Complete : Struct
         Header : Struct
            Header_CIP_Complete : Bool;
         END_STRUCT;
         "Chili Awetan" : Struct
            "T-02.00_CIP_Complete" : Bool;
            "T-03.00_CIP_Complete" : Bool;
            "T-04.00_CIP_Complete" : Bool;
         END_STRUCT;
         Tomato : Struct
            "T-05.00_CIP_Complete" : Bool;
         END_STRUCT;
         ChiliFresh : Struct
            "T-06.00_CIP_Complete" : Bool;
            "T-07.00_CIP_Complete" : Bool;
            "T-08.00_CIP_Complete" : Bool;
         END_STRUCT;
         Garlic : Struct
            "T-09.00_CIP_Complete" : Bool;
         END_STRUCT;
         Vinegar : Struct
            "T-10.00_CIP_Complete" : Bool;
         END_STRUCT;
         Homomixer : Struct
            "T-12.00_CIP_Complete" : Bool;
            "T-13.00_CIP_Complete" : Bool;
            "T-14.00_CIP_Complete" : Bool;
         END_STRUCT;
         "Blending Cluster 1" : Struct
            "T-20.00_CIP_Complete" : Bool;
            "T-21.00_CIP_Complete" : Bool;
            "T-30.00_CIP_Complete" : Bool;
            Blending_Cluster1_LineProduct_Complete : Bool;
            Free_CIP_Complete_1 : Bool;
            Free_CIP_Complete_2 : Bool;
         END_STRUCT;
         "Blending Cluster 2" : Struct
            "T-31.00_CIP_Complete" : Bool;
            "T-40.00_CIP_Complete" : Bool;
            "T-41.00_CIP_Complete" : Bool;
            Blending_Cluster2_LineProduct_Complete : Bool;
            Free_CIP_Complete_1 : Bool;
            Free_CIP_Complete_2 : Bool;
         END_STRUCT;
         "Rework Cluster 1" : Struct
            "T-22.00_CIP_Complete" : Bool;
         END_STRUCT;
         "Rework Cluster 2" : Struct
            "T-32.00_CIP_Complete" : Bool;
         END_STRUCT;
         "Buffer Cluster 1" : Struct
            "T-61.00_CIP_Complete" : Bool;
            "T-62.00_CIP_Complete" : Bool;
            "T61&T62_CIP_LineToPasteur_Complete" : Bool;
            "T-63.00_CIP_Complete" : Bool;
            "T-64.00_CIP_Complete" : Bool;
            "T63&T64_CIP_LineToPasteur_Complete" : Bool;
         END_STRUCT;
         "Buffer Cluster 2" : Struct
            "T-65.00_CIP_Complete" : Bool;
            "T-66.00_CIP_Complete" : Bool;
            "T65&T66_CIP_LineToPasteur_Complete" : Bool;
            "T-67.00_CIP_Complete" : Bool;
            "T-68.00_CIP_Complete" : Bool;
            "T67&T68_CIP_LineToPasteur_Complete" : Bool;
         END_STRUCT;
         "Storage THE 4" : Struct
            "T-23.00_CIP_Complete" : Bool;
            "T-24.00_CIP_Complete" : Bool;
            THE4_LineProduct_CIP_Complete : Bool;
         END_STRUCT;
         "Storage THE 5" : Struct
            "T-33.00_CIP_Tank_Complete" : Bool;
            "T-34.00_CIP_Tank_Complete" : Bool;
            "T33&T34_CIP_Line_Complete" : Bool;
            "T-35.00_CIP_Tank_Complete" : Bool;
            THE5_LineProduct_CIP_Complete : Bool;
         END_STRUCT;
         "T-79.00_CIP_Complete" : Bool;
         "T-81.00_CIP_Complete" : Bool;
         "T-84.00_CIP_Complete" : Bool;
         "T-85.00_CIP_Complete" : Bool;
         Free_CIP_Complete_5 : Bool;
         Free_CIP_Complete_6 : Bool;
         Free_CIP_Complete_7 : Bool;
         Free_CIP_Complete_8 : Bool;
         Free_CIP_Complete_9 : Bool;
         Free_CIP_Complete_10 : Bool;
         Free_CIP_Complete_11 : Bool;
         Free_CIP_Complete_12 : Bool;
         Free_CIP_Complete_13 : Bool;
         Free_CIP_Complete_14 : Bool;
         Free_CIP_Complete_15 : Bool;
         Free_CIP_Complete_16 : Bool;
         Osa_CIP_Complete : Bool;
         Free_CIP_Complete_18 : Bool;
         Free_CIP_Complete_19 : Bool;
         Free_CIP_Complete_20 : Bool;
         Free_CIP_Complete_21 : Bool;
         Free_CIP_Complete_22 : Bool;
         Free_CIP_Complete_23 : Bool;
         Free_CIP_Complete_24 : Bool;
      END_STRUCT;
   END_VAR
BEGIN
END_DATA_BLOCK

DATA_BLOCK "Mix_to_CIP"   // DB221
{ S7_Optimized_Access := 'FALSE' }
VERSION : 0.1
// stored: AutoNumber false, DBAccessibleFromOPCUA true, DBAccessibleFromWebserver true, IsOnlyStoredInLoadMemory false, IsWriteProtectedInAS false
   VAR
      HeartBeat : Bool := TRUE;
      CIP_Request : Struct
         Header : Struct
            Header_CIP_Request : Bool;
         END_STRUCT;
         "Chili Awetan" : Struct
            "T-02.00_CIP_Request" : Bool;
            "T-03.00_CIP_Request" : Bool;
            "T-04.00_CIP_Request" : Bool;
         END_STRUCT;
         Tomato : Struct
            "T-05.00_CIP_Request" : Bool;
         END_STRUCT;
         ChiliFresh : Struct
            "T-06.00_CIP_Request" : Bool;
            "T-07.00_CIP_Request" : Bool;
            "T-08.00_CIP_Request" : Bool;
         END_STRUCT;
         Garlic : Struct
            "T-09.00_CIP_Request" : Bool;
         END_STRUCT;
         Vinegar : Struct
            "T-10.00_CIP_Request" : Bool;
         END_STRUCT;
         Homomixer : Struct
            "T-12.00_CIP_Tank_Request" : Bool;
            "T-12.00_CIP_LineToBlend_Request" : Bool;
            "T-13.00_CIP_Tank_Request" : Bool;
            "T-13.00_CIP_LineToBlend_Request" : Bool;
            "T-14.00_CIP_Tank_Request" : Bool;
            "T-14.00_CIP_LineToBlend_Request" : Bool;
         END_STRUCT;
         "Blending Cluster 1" : Struct
            "T-20.00_CIP_Request" : Bool;
            "T-21.00_CIP_Request" : Bool;
            "T-30.00_CIP_Request" : Bool;
            Blending_Cluster1_LineProduct_Request : Bool;
            Free_CIP_Req_1 : Bool;
            Free_CIP_Req_2 : Bool;
         END_STRUCT;
         "Blending Cluster 2" : Struct
            "T-31.00_CIP_Request" : Bool;
            "T-40.00_CIP_Request" : Bool;
            "T-41.00_CIP_Request" : Bool;
            Blending_Cluster2_LineProduct_Request : Bool;
            Free_CIP_Req_1 : Bool;
            Free_CIP_Req_2 : Bool;
         END_STRUCT;
         "Rework Cluster 1" : Struct
            "T-22.00_CIP_Request" : Bool;
         END_STRUCT;
         "Rework Cluster 2" : Struct
            "T-32.00_CIP_Request" : Bool;
         END_STRUCT;
         "Buffer Cluster 1" : Struct
            "T-61.00_CIP_Request" : Bool;
            "T-62.00_CIP_Request" : Bool;
            "T61&T62_CIP_LineToPasteur_Request" : Bool;
            "T-63.00_CIP_Request" : Bool;
            "T-64.00_CIP_Request" : Bool;
            "T63&T64_CIP_LineToPasteur_Request" : Bool;
         END_STRUCT;
         "Buffer Cluster 2" : Struct
            "T-65.00_CIP_Request" : Bool;
            "T-66.00_CIP_Request" : Bool;
            "T65&T66_CIP_LineToPasteur_Request" : Bool;
            "T-67.00_CIP_Request" : Bool;
            "T-68.00_CIP_Request" : Bool;
            "T67&T68_CIP_LineToPasteur_Request" : Bool;
         END_STRUCT;
         "Storage THE 4" : Struct
            "T-23.00_CIP_Tank_Request" : Bool;
            "T-23.00_CIP_Line_Request" : Bool;
            "T-24.00_CIP_Tank_Request" : Bool;
            "T-24.00_CIP_Line_Request" : Bool;
            THE4_LineProduct_CIP_Request : Bool;
         END_STRUCT;
         "Storage THE 5" : Struct
            "T-33.00_CIP_Tank_Request" : Bool;
            "T-34.00_CIP_Tank_Request" : Bool;
            "T33&T34_CIP_Line_Request" : Bool;
            "T-35.00_CIP_Tank_Request" : Bool;
            "T-35.00_CIP_Line_Request" : Bool;
            THE5_LineProduct_CIP_Request : Bool;
         END_STRUCT;
         "T-79.00_CIP_Tank_Request" : Bool;
         "T-79.00_CIP_Line_Request" : Bool;
         "T-81.00_CIP_Request" : Bool;
         "T-84.00_CIP_Request" : Bool;
         "T-85.00_CIP_Request" : Bool;
         Free_CIP_Req_6 : Bool;
         Free_CIP_Req_7 : Bool;
         Free_CIP_Req_8 : Bool;
         Free_CIP_Req_9 : Bool;
         Free_CIP_Req_10 : Bool;
         Free_CIP_Req_11 : Bool;
         Free_CIP_Req_12 : Bool;
         Free_CIP_Req_13 : Bool;
         Free_CIP_Req_14 : Bool;
         Free_CIP_Req_15 : Bool;
         Free_CIP_Req_16 : Bool;
         Osa_CIP_Req : Bool;
         Free_CIP_Req_18 : Bool;
         Free_CIP_Req_19 : Bool;
         Free_CIP_Req_20 : Bool;
         Free_CIP_Req_21 : Bool;
         Free_CIP_Req_22 : Bool;
         Free_CIP_Req_23 : Bool;
         Free_CIP_Req_24 : Bool;
      END_STRUCT;
      CIP_Line_OK : Struct
         Header : Struct
            Header_CIP_LineOK : Bool;
         END_STRUCT;
         "Chili Awetan" : Struct
            "T-02.00_CIP_LineOK" : Bool;
            "T-03.00_CIP_LineOK" : Bool;
            "T-04.00_CIP_LineOK" : Bool;
         END_STRUCT;
         Tomato : Struct
            "T-05.00_CIP_LineOK" : Bool;
         END_STRUCT;
         ChiliFresh : Struct
            "T-06.00_CIP_LineOK" : Bool;
            "T-07.00_CIP_LineOK" : Bool;
            "T-08.00_CIP_LineOK" : Bool;
         END_STRUCT;
         Garlic : Struct
            "T-09.00_CIP_LineOK" : Bool;
         END_STRUCT;
         Vinegar : Struct
            "T-10.00_CIP_LineOK" : Bool;
         END_STRUCT;
         Homomixer : Struct
            "T-12.00_CIP_LineOK" : Bool;
            "T-13.00_CIP_LineOK" : Bool;
            "T-14.00_CIP_LineOK" : Bool;
         END_STRUCT;
         "Blending Cluster 1" : Struct
            "T-20.00_CIP_LineOK" : Bool;
            "T-21.00_CIP_LineOK" : Bool;
            "T-30.00_CIP_LineOK" : Bool;
            Blending_Cluster1_LineProduct_LineOK : Bool;
            Free_CIP_LineOK_1 : Bool;
            Free_CIP_LineOK_2 : Bool;
         END_STRUCT;
         "Blending Cluster 2" : Struct
            "T-31.00_CIP_LineOK" : Bool;
            "T-40.00_CIP_LineOK" : Bool;
            "T-41.00_CIP_LineOK" : Bool;
            Blending_Cluster2_LineProduct_LineOK : Bool;
            Free_CIP_LineOK_1 : Bool;
            Free_CIP_LineOK_2 : Bool;
         END_STRUCT;
         "Rework Cluster 1" : Struct
            "T-22.00_CIP_LineOK" : Bool;
         END_STRUCT;
         "Rework Cluster 2" : Struct
            "T-32.00_CIP_LineOK" : Bool;
         END_STRUCT;
         "Buffer Cluster 1" : Struct
            "T-61.00_CIP_LineOK" : Bool;
            "T-62.00_CIP_LineOK" : Bool;
            "T61&T62_CIP_LineToPasteur_LineOK" : Bool;
            "T-63.00_CIP_LineOK" : Bool;
            "T-64.00_CIP_LineOK" : Bool;
            "T63&T64_CIP_LineToPasteur_LineOK" : Bool;
         END_STRUCT;
         "Buffer Cluster 2" : Struct
            "T-65.00_CIP_LineOK" : Bool;
            "T-66.00_CIP_LineOK" : Bool;
            "T65&T66_CIP_LineToPasteur_LineOK" : Bool;
            "T-67.00_CIP_LineOK" : Bool;
            "T-68.00_CIP_LineOK" : Bool;
            "T67&T68_CIP_LineToPasteur_LineOK" : Bool;
         END_STRUCT;
         "Storage THE 4" : Struct
            "T-23.00_CIP_LineOK" : Bool;
            "T-24.00_CIP_LineOK" : Bool;
            THE4_LineProduct_CIP_LineOK : Bool;
         END_STRUCT;
         "Storage THE 5" : Struct
            "T-33.00_CIP_Tank_LineOK" : Bool;
            "T-34.00_CIP_Tank_LineOK" : Bool;
            "T33&T34_CIP_Line_LineOK" : Bool;
            "T-35.00_CIP_Tank_LineOK" : Bool;
            THE5_LineProduct_CIP_LineOK : Bool;
         END_STRUCT;
         "T-79.00_CIP_LineOK" : Bool;
         "T-81.00_CIP_LineOK" : Bool;
         "T-84.00_CIP_LineOK" : Bool;
         "T-85.00_CIP_LineOK" : Bool;
         Free_CIP_LineOK_5 : Bool;
         Free_CIP_LineOK_6 : Bool;
         Free_CIP_LineOK_7 : Bool;
         Free_CIP_LineOK_8 : Bool;
         Free_CIP_LineOK_9 : Bool;
         Free_CIP_LineOK_10 : Bool;
         Free_CIP_LineOK_11 : Bool;
         Free_CIP_LineOK_12 : Bool;
         Free_CIP_LineOK_13 : Bool;
         Free_CIP_LineOK_14 : Bool;
         Free_CIP_LineOK_15 : Bool;
         Free_CIP_LineOK_16 : Bool;
         Osa_CIP_LineOK : Bool;
         Free_CIP_LineOK_18 : Bool;
         Free_CIP_LineOK_19 : Bool;
         Free_CIP_LineOK_20 : Bool;
         Free_CIP_LineOK_21 : Bool;
         Free_CIP_LineOK_22 : Bool;
         Free_CIP_LineOK_23 : Bool;
         Free_CIP_LineOK_24 : Bool;
      END_STRUCT;
   END_VAR
BEGIN
END_DATA_BLOCK

DATA_BLOCK "Mix to PHE-2"   // DB404
{ S7_Optimized_Access := 'FALSE' }
VERSION : 0.1
// stored: AutoNumber false, DBAccessibleFromOPCUA true, DBAccessibleFromWebserver true, IsOnlyStoredInLoadMemory false, IsWriteProtectedInAS false
   VAR
      HeartBeat : Bool;
      Rework22_Porduct_Ready : Bool;
      Rework22_Transfer_On_Progress : Bool;
      "ST-11_Ready_Inload" : Bool;
      free_bool_5 : Bool;
      free_bool_6 : Bool;
      free_bool_7 : Bool;
      free_bool_8 : Bool;
      free_bool_9 : Bool;
      free_bool_10 : Bool;
      free_bool_11 : Bool;
      free_bool_12 : Bool;
      free_bool_13 : Bool;
      free_bool_14 : Bool;
      free_bool_15 : Bool;
      free_bool_16 : Bool;
      Level_Rework22 : Real;
      "Level_ST-11" : Real;
      free_real_3 : Real;
      free_real_4 : Real;
      free_real_5 : Real;
      free_real_6 : Real;
      free_real_7 : Real;
      free_real_8 : Real;
      free_real_9 : Real;
      free_real_10 : Real;
      free_real_11 : Real;
      free_real_12 : Real;
      free_real_13 : Real;
      free_real_14 : Real;
      free_real_15 : Real;
      free_real_16 : Real;
   END_VAR
BEGIN
END_DATA_BLOCK

DATA_BLOCK "PHE-2 to Mix"   // DB405
{ S7_Optimized_Access := 'FALSE' }
VERSION : 0.1
// stored: AutoNumber false, DBAccessibleFromOPCUA true, DBAccessibleFromWebserver true, IsOnlyStoredInLoadMemory false, IsWriteProtectedInAS false
   VAR
      Heartbeat : Bool;
      "High Level Coll Tank" : Bool;   // 1 = T-22 cant transfer to PHE-2
      "Alarm Prod" : Bool;   // 1 = Pause transfer from T-32 to PHE-2
      "CIP Request" : Bool;
      free_bool_5 : Bool;
      free_bool_6 : Bool;
      free_bool_7 : Bool;
      free_bool_8 : Bool;
      free_bool_9 : Bool;
      free_bool_10 : Bool;
      free_bool_11 : Bool;
      free_bool_12 : Bool;
      free_bool_13 : Bool;
      free_bool_14 : Bool;
      free_bool_15 : Bool;
      free_bool_16 : Bool;
      free_real_1 : Real;
      free_real_2 : Real;
      free_real_3 : Real;
      free_real_4 : Real;
      free_real_5 : Real;
      free_real_6 : Real;
      free_real_7 : Real;
      free_real_8 : Real;
      free_real_9 : Real;
      free_real_10 : Real;
      free_real_11 : Real;
      free_real_12 : Real;
      free_real_13 : Real;
      free_real_14 : Real;
      free_real_15 : Real;
      free_real_16 : Real;
   END_VAR
BEGIN
END_DATA_BLOCK

DATA_BLOCK "CIP to Osa"   // DB271
{ S7_Optimized_Access := 'FALSE' }
VERSION : 0.1
// stored: AutoNumber false, DBAccessibleFromOPCUA true, DBAccessibleFromWebserver true, IsOnlyStoredInLoadMemory false, IsWriteProtectedInAS false
   VAR
      HeartBeat : Bool;   // Clock 1Hz
      CIP_RequestOK : Bool;
      CIP_Transfer_inProg : Bool;
      CIP_Supply_ON : Bool;
      CIP_Complete : Bool;
      "CIP Prep MB on Process" : Bool;
      freeBool6 : Bool;
      freeBool7 : Bool;
      freeBool8 : Bool;
      freeBool9 : Bool;
      freeBool10 : Bool;
      freeBool11 : Bool;
      freeBool12 : Bool;
      freeBool13 : Bool;
      freeBool14 : Bool;
      freeBool15 : Bool;
   END_VAR
BEGIN
END_DATA_BLOCK

DATA_BLOCK "Osa to CIP"   // DB270
{ S7_Optimized_Access := 'FALSE' }
VERSION : 0.1
// stored: AutoNumber false, DBAccessibleFromOPCUA true, DBAccessibleFromWebserver true, IsOnlyStoredInLoadMemory false, IsWriteProtectedInAS false
   VAR
      HeartBeat : Bool;   // Clock 1Hz
      CIP_Request : Bool;
      CIP_LineOK : Bool;
      ObjectCIP : DWord;   // 3 : Blend, 19 : Tipper 1, 20 : Tipper 2
      "CIP OSA on Process" : Bool;
      freeBool5 : Bool;
      freeBool6 : Bool;
      freeBool7 : Bool;
      freeBool8 : Bool;
      freeBool9 : Bool;
      freeBool10 : Bool;
      freeBool11 : Bool;
      freeBool12 : Bool;
      freeBool13 : Bool;
      freeBool14 : Bool;
      freeBool15 : Bool;
   END_VAR
BEGIN
END_DATA_BLOCK

DATA_BLOCK "PHE-1 to Stock"   // DB407
{ S7_Optimized_Access := 'FALSE' }
VERSION : 0.1
// stored: AutoNumber false, DBAccessibleFromOPCUA true, DBAccessibleFromWebserver true, IsOnlyStoredInLoadMemory false, IsWriteProtectedInAS false
   VAR
      Heartbeat : Bool;
      CIP_Request : Bool;   // 1 = T-22 cant transfer to PHE-2
      free_bool_3 : Bool;   // 1 = Pause transfer from T-32 to PHE-2
      free_bool_4 : Bool;
      free_bool_5 : Bool;
      free_bool_6 : Bool;
      free_bool_7 : Bool;
      free_bool_8 : Bool;
      free_bool_9 : Bool;
      free_bool_10 : Bool;
      free_bool_11 : Bool;
      free_bool_12 : Bool;
      free_bool_13 : Bool;
      free_bool_14 : Bool;
      free_bool_15 : Bool;
      free_bool_16 : Bool;
      free_real_1 : Real;
      free_real_2 : Real;
      free_real_3 : Real;
      free_real_4 : Real;
      free_real_5 : Real;
      free_real_6 : Real;
      free_real_7 : Real;
      free_real_8 : Real;
      free_real_9 : Real;
      free_real_10 : Real;
      free_real_11 : Real;
      free_real_12 : Real;
      free_real_13 : Real;
      free_real_14 : Real;
      free_real_15 : Real;
      free_real_16 : Real;
   END_VAR
BEGIN
END_DATA_BLOCK

DATA_BLOCK "Stock to PHE-1"   // DB406
{ S7_Optimized_Access := 'FALSE' }
VERSION : 0.1
// stored: AutoNumber false, DBAccessibleFromOPCUA true, DBAccessibleFromWebserver true, IsOnlyStoredInLoadMemory false, IsWriteProtectedInAS false
   VAR
      HeartBeat : Bool;
      "ST-16_Ready_Inload" : Bool;
      free_bool_3 : Bool;
      free_bool_4 : Bool;
      free_bool_5 : Bool;
      free_bool_6 : Bool;
      free_bool_7 : Bool;
      free_bool_8 : Bool;
      free_bool_9 : Bool;
      free_bool_10 : Bool;
      free_bool_11 : Bool;
      free_bool_12 : Bool;
      free_bool_13 : Bool;
      free_bool_14 : Bool;
      free_bool_15 : Bool;
      free_bool_16 : Bool;
      "Level_ST-16" : Real;
      free_real_2 : Real;
      free_real_3 : Real;
      free_real_4 : Real;
      free_real_5 : Real;
      free_real_6 : Real;
      free_real_7 : Real;
      free_real_8 : Real;
      free_real_9 : Real;
      free_real_10 : Real;
      free_real_11 : Real;
      free_real_12 : Real;
      free_real_13 : Real;
      free_real_14 : Real;
      free_real_15 : Real;
      free_real_16 : Real;
   END_VAR
BEGIN
END_DATA_BLOCK

DATA_BLOCK "Mix_to_Salt"   // DB20
{ S7_Optimized_Access := 'FALSE' }
VERSION : 0.1
// stored: AutoNumber false, DBAccessibleFromOPCUA true, DBAccessibleFromWebserver true, IsOnlyStoredInLoadMemory false, IsWriteProtectedInAS false
   VAR
      Heartbeat : Bool;   // Alternating value of 0 and 1 to indicate that the PLC is alive
      Salt_Request : Bool;   // Customer calling for filling to mixer. Batching process will start after receive this signal
      Mixer_TankNum : Int;   // Customer to specify which mixer the transfer will go to (integer value 1 to 12 for mixer 1 to 12)
      "Weight SP" : Real;   // Customer to specify the total weight to batch
   END_VAR
BEGIN
END_DATA_BLOCK

DATA_BLOCK "Salt_to_Mix"   // DB21
{ S7_Optimized_Access := 'FALSE' }
VERSION : 0.1
// stored: AutoNumber true, DBAccessibleFromOPCUA true, DBAccessibleFromWebserver true, IsOnlyStoredInLoadMemory false, IsWriteProtectedInAS false
   VAR
      Heartbeat : Bool;   // Alternating value of 0 and 1 to indicate that the PLC is alive
      "System ready to run" : Bool;   // Gericke system is ready to receive signal from customer
      "Batching in process" : Bool;   // Signal received from customer, system is in batching process
      "Batching on hold" : Bool;   // Batching process on hold (either by alarm or manual hold by operator)
      "Batching completed" : Bool;   // Batching process completed, system will proceed to PTA transfer
      "Batching alarm" : Bool;   // Batching alarm exist (tolerance alarm, loadcell fault, etc)
      "PTA in process" : Bool;   // PTA transfer in process
      "PTA completed" : Bool;   // PTA transfer completed
      "PTA warning alarm" : Bool;   // PTA warning alarm exist (Conveying timeout, Filling timeout, etc)
      "PTA critical alarm" : Bool;   // Alarm exist (Overpressure, etc)
   END_VAR
BEGIN
END_DATA_BLOCK

DATA_BLOCK "Stock Tank Pouch"   // DB453
{ S7_Optimized_Access := 'FALSE' }
VERSION : 0.1
// stored: AutoNumber false, DBAccessibleFromOPCUA true, DBAccessibleFromWebserver true, IsOnlyStoredInLoadMemory false, IsWriteProtectedInAS false
   VAR RETAIN
      "ST-11 Product Request" : Bool;
      "ST-11 CIP Request" : Bool;
      "ST-14 Product Request" : Bool;
      "ST-14 CIP Request" : Bool;
      "ST-16 Product Request" : Bool;
      "ST-16 CIP Request" : Bool;
      "ST-11_P-81.01 Run" : Bool;
      "ST-14_P-84.01 Run" : Bool;
      "ST-14_P-84.02 Run" : Bool;
      "ST-16_P-82.01 Run" : Bool;
      "ST-14_P-84.01 SP" : Real;
      "ST-14_P-84.02 SP" : Real;
      "ST-16_P-82.01 SP" : Real;
      "ST-14_P-84.01 Act" : Real;
      "ST-14_P-84.02 Act" : Real;
      "ST-16_P-82.01 Act" : Real;
      "Level ST-14" : Real;
      "Level ST-16" : Real;
      "ST-11_P-81.01 SP" : Real;
      "ST-11_P-81.01 Act" : Real;
      "Level ST-11" : Real;
      freeReal12 : Real;
      freeReal13 : Real;
      freeReal14 : Real;
      freeReal15 : Real;
      freeReal16 : Real;
   END_VAR
BEGIN
END_DATA_BLOCK

DATA_BLOCK "Stock Tank to THE-1"   // DB451
{ S7_Optimized_Access := 'FALSE' }
VERSION : 0.1
// stored: AutoNumber false, DBAccessibleFromOPCUA true, DBAccessibleFromWebserver true, IsOnlyStoredInLoadMemory false, IsWriteProtectedInAS false
   VAR
      "ST-11_Ready_Inload" : Bool;
      "ST-16_Ready_Inload" : Bool;
      "ST-07_Ready_Inload" : Bool;
      "ST-09_Ready_Inload" : Bool;
      free_bool_5 : Bool;
      free_bool_6 : Bool;
      free_bool_7 : Bool;
      free_bool_8 : Bool;
      free_bool_9 : Bool;
      free_bool_10 : Bool;
      free_bool_11 : Bool;
      free_bool_12 : Bool;
      free_bool_13 : Bool;
      free_bool_14 : Bool;
      free_bool_15 : Bool;
      free_bool_16 : Bool;
      "Level_ST-11" : Real;
      "Level_ST-16" : Real;
      "Level_ST-07" : Real;
      "Level_ST-09" : Real;
      free_real_5 : Real;
      free_real_6 : Real;
      free_real_7 : Real;
      free_real_8 : Real;
      free_byte_1 : Byte;
      free_byte_2 : Byte;
      free_byte_3 : Byte;
      free_byte_4 : Byte;
      free_byte_5 : Byte;
      free_byte_6 : Byte;
      free_byte_7 : Byte;
      free_byte_8 : Byte;
   END_VAR
BEGIN
END_DATA_BLOCK

DATA_BLOCK "THE-1 to Stock Tank"   // DB452
{ S7_Optimized_Access := 'FALSE' }
VERSION : 0.1
// stored: AutoNumber false, DBAccessibleFromOPCUA true, DBAccessibleFromWebserver true, IsOnlyStoredInLoadMemory false, IsWriteProtectedInAS false
   VAR
      CIP_Request : Bool;
      free_bool_2 : Bool;
      free_bool_3 : Bool;
      free_bool_4 : Bool;
      free_bool_5 : Bool;
      free_bool_6 : Bool;
      free_bool_7 : Bool;
      free_bool_8 : Bool;
      free_bool_9 : Bool;
      free_bool_10 : Bool;
      free_bool_11 : Bool;
      free_bool_12 : Bool;
      free_bool_13 : Bool;
      free_bool_14 : Bool;
      free_bool_15 : Bool;
      free_bool_16 : Bool;
      free_real_1 : Real;
      free_real_2 : Real;
      free_real_3 : Real;
      free_real_4 : Real;
      free_real_5 : Real;
      free_real_6 : Real;
      free_real_7 : Real;
      free_real_8 : Real;
      free_byte_1 : Byte;
      free_byte_2 : Byte;
      free_byte_3 : Byte;
      free_byte_4 : Byte;
      free_byte_5 : Byte;
      free_byte_6 : Byte;
      free_byte_7 : Byte;
      free_byte_8 : Byte;
   END_VAR
BEGIN
END_DATA_BLOCK

DATA_BLOCK "Mix to Sugar"   // DB230
{ S7_Optimized_Access := 'FALSE' }
VERSION : 0.1
// stored: AutoNumber false, DBAccessibleFromOPCUA true, DBAccessibleFromWebserver true, IsOnlyStoredInLoadMemory false, IsWriteProtectedInAS false
   VAR
      HeartBeat : Bool;   // Alternating value of 0 and 1 to indicate that the PLC is alive
      "Mixer system call for filling" : Bool;   // Customer calling for filling to mixer. Transfer process will start after receive this signal
      "Target mixer" : Int;   // Customer to specify which mixer the transfer will go to (integer value 1 to 12 for mixer 1 to 12)
      "Weight setpoint for mixer" : Real;   // Customer to specify the total weight to batch
   END_VAR
BEGIN
END_DATA_BLOCK

DATA_BLOCK "Sugar to Mix"   // DB231
{ S7_Optimized_Access := 'FALSE' }
VERSION : 0.1
// stored: AutoNumber false, DBAccessibleFromOPCUA true, DBAccessibleFromWebserver true, IsOnlyStoredInLoadMemory false, IsWriteProtectedInAS false
   VAR
      HeartBeat : Bool;   // Alternating value of 0 and 1 to indicate that the PLC is alive
      "System ready to run" : Bool;   // Scala system is ready to receive signal from customer
      "Transfer in process" : Bool;   // transfer in process
      "Transfer completed" : Bool;   // transfer completed
      "Transfer alarm" : Bool;   // warning alarm exist (Conveying timeout, Filling timeout, etc)
      "Weight Actual for Mixer" : Real;
   END_VAR
BEGIN
END_DATA_BLOCK

DATA_BLOCK "T-32 to THE-1"   // DB401
{ S7_Optimized_Access := 'FALSE' }
VERSION : 0.1
// stored: AutoNumber false, DBAccessibleFromOPCUA true, DBAccessibleFromWebserver true, IsOnlyStoredInLoadMemory false, IsWriteProtectedInAS false
   VAR
      Porduct_Ready : Bool;
      Transfer_On_Progress : Bool;
      free_bool_3 : Bool;
      free_bool_4 : Bool;
      free_bool_5 : Bool;
      free_bool_6 : Bool;
      free_bool_7 : Bool;
      free_bool_8 : Bool;
      free_bool_9 : Bool;
      free_bool_10 : Bool;
      free_bool_11 : Bool;
      free_bool_12 : Bool;
      free_bool_13 : Bool;
      free_bool_14 : Bool;
      free_bool_15 : Bool;
      free_bool_16 : Bool;
      Level_Tank : Real;
      free_real_2 : Real;
      free_real_3 : Real;
      free_real_4 : Real;
      free_real_5 : Real;
      free_real_6 : Real;
      free_real_7 : Real;
      free_real_8 : Real;
      free_byte_1 : Byte;
      free_byte_2 : Byte;
      free_byte_3 : Byte;
      free_byte_4 : Byte;
      free_byte_5 : Byte;
      free_byte_6 : Byte;
      free_byte_7 : Byte;
      free_byte_8 : Byte;
   END_VAR
BEGIN
END_DATA_BLOCK

DATA_BLOCK "THE-1 to T-32"   // DB402
{ S7_Optimized_Access := 'FALSE' }
VERSION : 0.1
// stored: AutoNumber false, DBAccessibleFromOPCUA true, DBAccessibleFromWebserver true, IsOnlyStoredInLoadMemory false, IsWriteProtectedInAS false
   VAR
      "High Level Coll Tank" : Bool;   // 1 = T-32 cant transfer to THE-1
      "Alarm Prod" : Bool;   // 1 = Pause transfer from T-32 to THE-1
      free_bool_3 : Bool;
      free_bool_4 : Bool;
      free_bool_5 : Bool;
      free_bool_6 : Bool;
      free_bool_7 : Bool;
      free_bool_8 : Bool;
      free_bool_9 : Bool;
      free_bool_10 : Bool;
      free_bool_11 : Bool;
      free_bool_12 : Bool;
      free_bool_13 : Bool;
      free_bool_14 : Bool;
      free_bool_15 : Bool;
      free_bool_16 : Bool;
      free_real_1 : Real;
      free_real_2 : Real;
      free_real_3 : Real;
      free_real_4 : Real;
      free_real_5 : Real;
      free_real_6 : Real;
      free_real_7 : Real;
      free_real_8 : Real;
      free_byte_1 : Byte;
      free_byte_2 : Byte;
      free_byte_3 : Byte;
      free_byte_4 : Byte;
      free_byte_5 : Byte;
      free_byte_6 : Byte;
      free_byte_7 : Byte;
      free_byte_8 : Byte;
   END_VAR
BEGIN
END_DATA_BLOCK

DATA_BLOCK "MB to Tipper1"   // DB245
{ S7_Optimized_Access := 'FALSE' }
VERSION : 0.1
// stored: AutoNumber false, DBAccessibleFromOPCUA true, DBAccessibleFromWebserver true, IsOnlyStoredInLoadMemory false, IsWriteProtectedInAS false
   VAR
      HeartBeat : Bool;   // Clock 1Hz
      Product_Request : Bool;
      Product_Line_OK : Bool;
      freeBool3 : Bool;
      freeBool4 : Bool;
      freeBool5 : Bool;
      freeBool6 : Bool;
      freeBool7 : Bool;
      freeBool8 : Bool;
      freeBool9 : Bool;
      freeBool10 : Bool;
      freeBool11 : Bool;
      freeBool12 : Bool;
      freeBool13 : Bool;
      freeBool14 : Bool;
      freeBool15 : Bool;
      freeBool16 : Bool;
      freeBool17 : Bool;
      freeBool18 : Bool;
      freeBool19 : Bool;
      freeBool20 : Bool;
      freeBool21 : Bool;
      freeBool22 : Bool;
      freeBool23 : Bool;
   END_VAR
BEGIN
END_DATA_BLOCK

DATA_BLOCK "Tipper1 to MB"   // DB244
{ S7_Optimized_Access := 'FALSE' }
VERSION : 0.1
// stored: AutoNumber false, DBAccessibleFromOPCUA true, DBAccessibleFromWebserver true, IsOnlyStoredInLoadMemory false, IsWriteProtectedInAS false
   VAR
      HeartBeat : Bool;   // Clock 1hz
      Product_Ready : Bool;
      Product_LineOpen : Bool;
      Product_SupplyON : Bool;
      Product_Transfer_Complete : Bool;
      freeBool5 : Bool;
      freeBool6 : Bool;
      freeBool7 : Bool;
      freeBool8 : Bool;
      freeBool9 : Bool;
      freeBool10 : Bool;
      freeBool11 : Bool;
      freeBool12 : Bool;
      freeBool13 : Bool;
      freeBool14 : Bool;
      freeBool15 : Bool;
      freeBool16 : Bool;
      freeBool17 : Bool;
      freeBool18 : Bool;
      freeBool19 : Bool;
      freeBool20 : Bool;
      freeBool21 : Bool;
      freeBool22 : Bool;
      freeBool23 : Bool;
   END_VAR
BEGIN
END_DATA_BLOCK

DATA_BLOCK "MB to Tipper2"   // DB241
{ S7_Optimized_Access := 'FALSE' }
VERSION : 0.1
// stored: AutoNumber false, DBAccessibleFromOPCUA true, DBAccessibleFromWebserver true, IsOnlyStoredInLoadMemory false, IsWriteProtectedInAS false
   VAR
      HeartBeat : Bool;   // Clock 1Hz
      Product_Request : Bool;
      Product_Line_OK : Bool;
      freeBool3 : Bool;
      freeBool4 : Bool;
      freeBool5 : Bool;
      freeBool6 : Bool;
      freeBool7 : Bool;
      freeBool8 : Bool;
      freeBool9 : Bool;
      freeBool10 : Bool;
      freeBool11 : Bool;
      freeBool12 : Bool;
      freeBool13 : Bool;
      freeBool14 : Bool;
      freeBool15 : Bool;
      freeBool16 : Bool;
      freeBool17 : Bool;
      freeBool18 : Bool;
      freeBool19 : Bool;
      freeBool20 : Bool;
      freeBool21 : Bool;
      freeBool22 : Bool;
      freeBool23 : Bool;
   END_VAR
BEGIN
END_DATA_BLOCK

DATA_BLOCK "Tipper2 to MB"   // DB240
{ S7_Optimized_Access := 'FALSE' }
VERSION : 0.1
// stored: AutoNumber false, DBAccessibleFromOPCUA true, DBAccessibleFromWebserver true, IsOnlyStoredInLoadMemory false, IsWriteProtectedInAS false
   VAR
      HeartBeat : Bool;   // Clock 1hz
      Product_Ready : Bool;
      Product_LineOpen : Bool;
      Product_SupplyON : Bool;
      Product_Transfer_Complete : Bool;
      freeBool5 : Bool;
      freeBool6 : Bool;
      freeBool7 : Bool;
      freeBool8 : Bool;
      freeBool9 : Bool;
      freeBool10 : Bool;
      freeBool11 : Bool;
      freeBool12 : Bool;
      freeBool13 : Bool;
      freeBool14 : Bool;
      freeBool15 : Bool;
      freeBool16 : Bool;
      freeBool17 : Bool;
      freeBool18 : Bool;
      freeBool19 : Bool;
      freeBool20 : Bool;
      freeBool21 : Bool;
      freeBool22 : Bool;
      freeBool23 : Bool;
   END_VAR
BEGIN
END_DATA_BLOCK

DATA_BLOCK "Blend to Preparation"   // DB461
{ S7_Optimized_Access := 'TRUE' }
VERSION : 0.1
// stored: AutoNumber false, DBAccessibleFromOPCUA true, DBAccessibleFromWebserver true, IsOnlyStoredInLoadMemory false, IsRetainMemResEnabled false, IsWriteProtectedInAS false, MemoryReserve 0
   VAR
      "T-20" : Struct
         Raw_Material : Struct
            HW : Struct
               DoseRun : Bool;
               DoseHeld : Bool;
               DoseComplete : Bool;
               ValveCMD : Bool;
               PumpCMD : Bool;
               Header1_Req : Bool;
               Header2_Req : Bool;
            END_STRUCT;
            ChiliAwetan_1 : Struct
               DoseRun : Bool;
               DoseHeld : Bool;
               DoseComplete : Bool;
               ValveCMD : Bool;
               PumpCMD : Bool;
               Header1_Req : Bool;
               Header2_Req : Bool;
            END_STRUCT;
            ChiliAwetan_2 : Struct
               DoseRun : Bool;
               DoseHeld : Bool;
               DoseComplete : Bool;
               ValveCMD : Bool;
               PumpCMD : Bool;
               Header1_Req : Bool;
               Header2_Req : Bool;
            END_STRUCT;
            ChiliAwetan_3 : Struct
               DoseRun : Bool;
               DoseHeld : Bool;
               DoseComplete : Bool;
               ValveCMD : Bool;
               PumpCMD : Bool;
               Header1_Req : Bool;
               Header2_Req : Bool;
            END_STRUCT;
            Tomato : Struct
               DoseRun : Bool;
               DoseHeld : Bool;
               DoseComplete : Bool;
               ValveCMD : Bool;
               PumpCMD : Bool;
               Header1_Req : Bool;
               Header2_Req : Bool;
            END_STRUCT;
            ChiliFresh_1 : Struct
               DoseRun : Bool;
               DoseHeld : Bool;
               DoseComplete : Bool;
               ValveCMD : Bool;
               PumpCMD : Bool;
               Header1_Req : Bool;
               Header2_Req : Bool;
            END_STRUCT;
            ChiliFresh_2 : Struct
               DoseRun : Bool;
               DoseHeld : Bool;
               DoseComplete : Bool;
               ValveCMD : Bool;
               PumpCMD : Bool;
               Header1_Req : Bool;
               Header2_Req : Bool;
            END_STRUCT;
            ChiliFresh_3 : Struct
               DoseRun : Bool;
               DoseHeld : Bool;
               DoseComplete : Bool;
               ValveCMD : Bool;
               PumpCMD : Bool;
               Header1_Req : Bool;
               Header2_Req : Bool;
            END_STRUCT;
            Garlic : Struct
               DoseRun : Bool;
               DoseHeld : Bool;
               DoseComplete : Bool;
               ValveCMD : Bool;
               PumpCMD : Bool;
               Header1_Req : Bool;
               Header2_Req : Bool;
            END_STRUCT;
            Vinegar : Struct
               DoseRun : Bool;
               DoseHeld : Bool;
               DoseComplete : Bool;
               ValveCMD : Bool;
               PumpCMD : Bool;
               Header1_Req : Bool;
               Header2_Req : Bool;
            END_STRUCT;
         END_STRUCT;
         LineHeader1_OK : Bool;
         LineHeader2_OK : Bool;
         LineVinegar_OK : Bool;
         freeBool_4 : Bool;
         freeBool_5 : Bool;
         freeReal_1 : Bool;
         freeReal_2 : Bool;
         freeReal_3 : Bool;
         freeReal_4 : Bool;
         freeReal_5 : Bool;
      END_STRUCT;
      "T-21" : Struct
         Raw_Material : Struct
            HW : Struct
               DoseRun : Bool;
               DoseHeld : Bool;
               DoseComplete : Bool;
               ValveCMD : Bool;
               PumpCMD : Bool;
               Header1_Req : Bool;
               Header2_Req : Bool;
            END_STRUCT;
            ChiliAwetan_1 : Struct
               DoseRun : Bool;
               DoseHeld : Bool;
               DoseComplete : Bool;
               ValveCMD : Bool;
               PumpCMD : Bool;
               Header1_Req : Bool;
               Header2_Req : Bool;
            END_STRUCT;
            ChiliAwetan_2 : Struct
               DoseRun : Bool;
               DoseHeld : Bool;
               DoseComplete : Bool;
               ValveCMD : Bool;
               PumpCMD : Bool;
               Header1_Req : Bool;
               Header2_Req : Bool;
            END_STRUCT;
            ChiliAwetan_3 : Struct
               DoseRun : Bool;
               DoseHeld : Bool;
               DoseComplete : Bool;
               ValveCMD : Bool;
               PumpCMD : Bool;
               Header1_Req : Bool;
               Header2_Req : Bool;
            END_STRUCT;
            Tomato : Struct
               DoseRun : Bool;
               DoseHeld : Bool;
               DoseComplete : Bool;
               ValveCMD : Bool;
               PumpCMD : Bool;
               Header1_Req : Bool;
               Header2_Req : Bool;
            END_STRUCT;
            ChiliFresh_1 : Struct
               DoseRun : Bool;
               DoseHeld : Bool;
               DoseComplete : Bool;
               ValveCMD : Bool;
               PumpCMD : Bool;
               Header1_Req : Bool;
               Header2_Req : Bool;
            END_STRUCT;
            ChiliFresh_2 : Struct
               DoseRun : Bool;
               DoseHeld : Bool;
               DoseComplete : Bool;
               ValveCMD : Bool;
               PumpCMD : Bool;
               Header1_Req : Bool;
               Header2_Req : Bool;
            END_STRUCT;
            ChiliFresh_3 : Struct
               DoseRun : Bool;
               DoseHeld : Bool;
               DoseComplete : Bool;
               ValveCMD : Bool;
               PumpCMD : Bool;
               Header1_Req : Bool;
               Header2_Req : Bool;
            END_STRUCT;
            Garlic : Struct
               DoseRun : Bool;
               DoseHeld : Bool;
               DoseComplete : Bool;
               ValveCMD : Bool;
               PumpCMD : Bool;
               Header1_Req : Bool;
               Header2_Req : Bool;
            END_STRUCT;
            Vinegar : Struct
               DoseRun : Bool;
               DoseHeld : Bool;
               DoseComplete : Bool;
               ValveCMD : Bool;
               PumpCMD : Bool;
               Header1_Req : Bool;
               Header2_Req : Bool;
            END_STRUCT;
         END_STRUCT;
         LineHeader1_OK : Bool;
         LineHeader2_OK : Bool;
         LineVinegar_OK : Bool;
         freeBool_4 : Bool;
         freeBool_5 : Bool;
         freeReal_1 : Bool;
         freeReal_2 : Bool;
         freeReal_3 : Bool;
         freeReal_4 : Bool;
         freeReal_5 : Bool;
      END_STRUCT;
      "T-30" : Struct
         Raw_Material : Struct
            HW : Struct
               DoseRun : Bool;
               DoseHeld : Bool;
               DoseComplete : Bool;
               ValveCMD : Bool;
               PumpCMD : Bool;
               Header1_Req : Bool;
               Header2_Req : Bool;
            END_STRUCT;
            ChiliAwetan_1 : Struct
               DoseRun : Bool;
               DoseHeld : Bool;
               DoseComplete : Bool;
               ValveCMD : Bool;
               PumpCMD : Bool;
               Header1_Req : Bool;
               Header2_Req : Bool;
            END_STRUCT;
            ChiliAwetan_2 : Struct
               DoseRun : Bool;
               DoseHeld : Bool;
               DoseComplete : Bool;
               ValveCMD : Bool;
               PumpCMD : Bool;
               Header1_Req : Bool;
               Header2_Req : Bool;
            END_STRUCT;
            ChiliAwetan_3 : Struct
               DoseRun : Bool;
               DoseHeld : Bool;
               DoseComplete : Bool;
               ValveCMD : Bool;
               PumpCMD : Bool;
               Header1_Req : Bool;
               Header2_Req : Bool;
            END_STRUCT;
            Tomato : Struct
               DoseRun : Bool;
               DoseHeld : Bool;
               DoseComplete : Bool;
               ValveCMD : Bool;
               PumpCMD : Bool;
               Header1_Req : Bool;
               Header2_Req : Bool;
            END_STRUCT;
            ChiliFresh_1 : Struct
               DoseRun : Bool;
               DoseHeld : Bool;
               DoseComplete : Bool;
               ValveCMD : Bool;
               PumpCMD : Bool;
               Header1_Req : Bool;
               Header2_Req : Bool;
            END_STRUCT;
            ChiliFresh_2 : Struct
               DoseRun : Bool;
               DoseHeld : Bool;
               DoseComplete : Bool;
               ValveCMD : Bool;
               PumpCMD : Bool;
               Header1_Req : Bool;
               Header2_Req : Bool;
            END_STRUCT;
            ChiliFresh_3 : Struct
               DoseRun : Bool;
               DoseHeld : Bool;
               DoseComplete : Bool;
               ValveCMD : Bool;
               PumpCMD : Bool;
               Header1_Req : Bool;
               Header2_Req : Bool;
            END_STRUCT;
            Garlic : Struct
               DoseRun : Bool;
               DoseHeld : Bool;
               DoseComplete : Bool;
               ValveCMD : Bool;
               PumpCMD : Bool;
               Header1_Req : Bool;
               Header2_Req : Bool;
            END_STRUCT;
            Vinegar : Struct
               DoseRun : Bool;
               DoseHeld : Bool;
               DoseComplete : Bool;
               ValveCMD : Bool;
               PumpCMD : Bool;
               Header1_Req : Bool;
               Header2_Req : Bool;
            END_STRUCT;
         END_STRUCT;
         LineHeader1_OK : Bool;
         LineHeader2_OK : Bool;
         LineVinegar_OK : Bool;
         freeBool_4 : Bool;
         freeBool_5 : Bool;
         freeReal_1 : Bool;
         freeReal_2 : Bool;
         freeReal_3 : Bool;
         freeReal_4 : Bool;
         freeReal_5 : Bool;
      END_STRUCT;
      "T-31" : Struct
         Raw_Material : Struct
            HW : Struct
               DoseRun : Bool;
               DoseHeld : Bool;
               DoseComplete : Bool;
               ValveCMD : Bool;
               PumpCMD : Bool;
               Header1_Req : Bool;
               Header2_Req : Bool;
            END_STRUCT;
            ChiliAwetan_1 : Struct
               DoseRun : Bool;
               DoseHeld : Bool;
               DoseComplete : Bool;
               ValveCMD : Bool;
               PumpCMD : Bool;
               Header1_Req : Bool;
               Header2_Req : Bool;
            END_STRUCT;
            ChiliAwetan_2 : Struct
               DoseRun : Bool;
               DoseHeld : Bool;
               DoseComplete : Bool;
               ValveCMD : Bool;
               PumpCMD : Bool;
               Header1_Req : Bool;
               Header2_Req : Bool;
            END_STRUCT;
            ChiliAwetan_3 : Struct
               DoseRun : Bool;
               DoseHeld : Bool;
               DoseComplete : Bool;
               ValveCMD : Bool;
               PumpCMD : Bool;
               Header1_Req : Bool;
               Header2_Req : Bool;
            END_STRUCT;
            Tomato : Struct
               DoseRun : Bool;
               DoseHeld : Bool;
               DoseComplete : Bool;
               ValveCMD : Bool;
               PumpCMD : Bool;
               Header1_Req : Bool;
               Header2_Req : Bool;
            END_STRUCT;
            ChiliFresh_1 : Struct
               DoseRun : Bool;
               DoseHeld : Bool;
               DoseComplete : Bool;
               ValveCMD : Bool;
               PumpCMD : Bool;
               Header1_Req : Bool;
               Header2_Req : Bool;
            END_STRUCT;
            ChiliFresh_2 : Struct
               DoseRun : Bool;
               DoseHeld : Bool;
               DoseComplete : Bool;
               ValveCMD : Bool;
               PumpCMD : Bool;
               Header1_Req : Bool;
               Header2_Req : Bool;
            END_STRUCT;
            ChiliFresh_3 : Struct
               DoseRun : Bool;
               DoseHeld : Bool;
               DoseComplete : Bool;
               ValveCMD : Bool;
               PumpCMD : Bool;
               Header1_Req : Bool;
               Header2_Req : Bool;
            END_STRUCT;
            Garlic : Struct
               DoseRun : Bool;
               DoseHeld : Bool;
               DoseComplete : Bool;
               ValveCMD : Bool;
               PumpCMD : Bool;
               Header1_Req : Bool;
               Header2_Req : Bool;
            END_STRUCT;
            Vinegar : Struct
               DoseRun : Bool;
               DoseHeld : Bool;
               DoseComplete : Bool;
               ValveCMD : Bool;
               PumpCMD : Bool;
               Header1_Req : Bool;
               Header2_Req : Bool;
            END_STRUCT;
         END_STRUCT;
         LineHeader1_OK : Bool;
         LineHeader2_OK : Bool;
         LineVinegar_OK : Bool;
         freeBool_4 : Bool;
         freeBool_5 : Bool;
         freeReal_1 : Bool;
         freeReal_2 : Bool;
         freeReal_3 : Bool;
         freeReal_4 : Bool;
         freeReal_5 : Bool;
      END_STRUCT;
      "T-40" : Struct
         Raw_Material : Struct
            HW : Struct
               DoseRun : Bool;
               DoseHeld : Bool;
               DoseComplete : Bool;
               ValveCMD : Bool;
               PumpCMD : Bool;
               Header1_Req : Bool;
               Header2_Req : Bool;
            END_STRUCT;
            ChiliAwetan_1 : Struct
               DoseRun : Bool;
               DoseHeld : Bool;
               DoseComplete : Bool;
               ValveCMD : Bool;
               PumpCMD : Bool;
               Header1_Req : Bool;
               Header2_Req : Bool;
            END_STRUCT;
            ChiliAwetan_2 : Struct
               DoseRun : Bool;
               DoseHeld : Bool;
               DoseComplete : Bool;
               ValveCMD : Bool;
               PumpCMD : Bool;
               Header1_Req : Bool;
               Header2_Req : Bool;
            END_STRUCT;
            ChiliAwetan_3 : Struct
               DoseRun : Bool;
               DoseHeld : Bool;
               DoseComplete : Bool;
               ValveCMD : Bool;
               PumpCMD : Bool;
               Header1_Req : Bool;
               Header2_Req : Bool;
            END_STRUCT;
            Tomato : Struct
               DoseRun : Bool;
               DoseHeld : Bool;
               DoseComplete : Bool;
               ValveCMD : Bool;
               PumpCMD : Bool;
               Header1_Req : Bool;
               Header2_Req : Bool;
            END_STRUCT;
            ChiliFresh_1 : Struct
               DoseRun : Bool;
               DoseHeld : Bool;
               DoseComplete : Bool;
               ValveCMD : Bool;
               PumpCMD : Bool;
               Header1_Req : Bool;
               Header2_Req : Bool;
            END_STRUCT;
            ChiliFresh_2 : Struct
               DoseRun : Bool;
               DoseHeld : Bool;
               DoseComplete : Bool;
               ValveCMD : Bool;
               PumpCMD : Bool;
               Header1_Req : Bool;
               Header2_Req : Bool;
            END_STRUCT;
            ChiliFresh_3 : Struct
               DoseRun : Bool;
               DoseHeld : Bool;
               DoseComplete : Bool;
               ValveCMD : Bool;
               PumpCMD : Bool;
               Header1_Req : Bool;
               Header2_Req : Bool;
            END_STRUCT;
            Garlic : Struct
               DoseRun : Bool;
               DoseHeld : Bool;
               DoseComplete : Bool;
               ValveCMD : Bool;
               PumpCMD : Bool;
               Header1_Req : Bool;
               Header2_Req : Bool;
            END_STRUCT;
            Vinegar : Struct
               DoseRun : Bool;
               DoseHeld : Bool;
               DoseComplete : Bool;
               ValveCMD : Bool;
               PumpCMD : Bool;
               Header1_Req : Bool;
               Header2_Req : Bool;
            END_STRUCT;
         END_STRUCT;
         LineHeader1_OK : Bool;
         LineHeader2_OK : Bool;
         LineVinegar_OK : Bool;
         freeBool_4 : Bool;
         freeBool_5 : Bool;
         freeReal_1 : Bool;
         freeReal_2 : Bool;
         freeReal_3 : Bool;
         freeReal_4 : Bool;
         freeReal_5 : Bool;
      END_STRUCT;
      "T-41" : Struct
         Raw_Material : Struct
            HW : Struct
               DoseRun : Bool;
               DoseHeld : Bool;
               DoseComplete : Bool;
               ValveCMD : Bool;
               PumpCMD : Bool;
               Header1_Req : Bool;
               Header2_Req : Bool;
            END_STRUCT;
            ChiliAwetan_1 : Struct
               DoseRun : Bool;
               DoseHeld : Bool;
               DoseComplete : Bool;
               ValveCMD : Bool;
               PumpCMD : Bool;
               Header1_Req : Bool;
               Header2_Req : Bool;
            END_STRUCT;
            ChiliAwetan_2 : Struct
               DoseRun : Bool;
               DoseHeld : Bool;
               DoseComplete : Bool;
               ValveCMD : Bool;
               PumpCMD : Bool;
               Header1_Req : Bool;
               Header2_Req : Bool;
            END_STRUCT;
            ChiliAwetan_3 : Struct
               DoseRun : Bool;
               DoseHeld : Bool;
               DoseComplete : Bool;
               ValveCMD : Bool;
               PumpCMD : Bool;
               Header1_Req : Bool;
               Header2_Req : Bool;
            END_STRUCT;
            Tomato : Struct
               DoseRun : Bool;
               DoseHeld : Bool;
               DoseComplete : Bool;
               ValveCMD : Bool;
               PumpCMD : Bool;
               Header1_Req : Bool;
               Header2_Req : Bool;
            END_STRUCT;
            ChiliFresh_1 : Struct
               DoseRun : Bool;
               DoseHeld : Bool;
               DoseComplete : Bool;
               ValveCMD : Bool;
               PumpCMD : Bool;
               Header1_Req : Bool;
               Header2_Req : Bool;
            END_STRUCT;
            ChiliFresh_2 : Struct
               DoseRun : Bool;
               DoseHeld : Bool;
               DoseComplete : Bool;
               ValveCMD : Bool;
               PumpCMD : Bool;
               Header1_Req : Bool;
               Header2_Req : Bool;
            END_STRUCT;
            ChiliFresh_3 : Struct
               DoseRun : Bool;
               DoseHeld : Bool;
               DoseComplete : Bool;
               ValveCMD : Bool;
               PumpCMD : Bool;
               Header1_Req : Bool;
               Header2_Req : Bool;
            END_STRUCT;
            Garlic : Struct
               DoseRun : Bool;
               DoseHeld : Bool;
               DoseComplete : Bool;
               ValveCMD : Bool;
               PumpCMD : Bool;
               Header1_Req : Bool;
               Header2_Req : Bool;
            END_STRUCT;
            Vinegar : Struct
               DoseRun : Bool;
               DoseHeld : Bool;
               DoseComplete : Bool;
               ValveCMD : Bool;
               PumpCMD : Bool;
               Header1_Req : Bool;
               Header2_Req : Bool;
            END_STRUCT;
         END_STRUCT;
         LineHeader1_OK : Bool;
         LineHeader2_OK : Bool;
         LineVinegar_OK : Bool;
         freeBool_4 : Bool;
         freeBool_5 : Bool;
         freeReal_1 : Bool;
         freeReal_2 : Bool;
         freeReal_3 : Bool;
         freeReal_4 : Bool;
         freeReal_5 : Bool;
      END_STRUCT;
   END_VAR
   VAR RETAIN
      Recipe : Struct
         "T-20" : Struct
            HW : Struct
               Sp_Flush_to_BlendQty : Real;
               Sp_Flush_to_DrainQty : Real;
               Sp_DrainTime : DInt;
               SP_PumpSpeed : Real;
            END_STRUCT;
            ChiliAwetan_1 : Struct
               Sp_DoseQty : Real;
               SP_PumpSpeed : Real;
            END_STRUCT;
            ChiliAwetan_2 : Struct
               Sp_DoseQty : Real;
               SP_PumpSpeed : Real;
            END_STRUCT;
            ChiliAwetan_3 : Struct
               Sp_DoseQty : Real;
               SP_PumpSpeed : Real;
            END_STRUCT;
            Tomato : Struct
               Sp_DoseQty : Real;
               SP_PumpSpeed : Real;
            END_STRUCT;
            ChiliFresh_1 : Struct
               Sp_DoseQty : Real;
               SP_PumpSpeed : Real;
            END_STRUCT;
            ChiliFresh_2 : Struct
               Sp_DoseQty : Real;
               SP_PumpSpeed : Real;
            END_STRUCT;
            ChiliFresh_3 : Struct
               Sp_DoseQty : Real;
               SP_PumpSpeed : Real;
            END_STRUCT;
            Garlic : Struct
               Sp_DoseQty : Real;
               SP_PumpSpeed : Real;
            END_STRUCT;
            Vinegar : Struct
               Sp_DoseQty : Real;
               SP_PumpSpeed : Real;
            END_STRUCT;
            Sugar : Struct
               Sp_DoseQty : Real;
               SP_PumpSpeed : Real;
            END_STRUCT;
            Salt : Struct
               Sp_DoseQty : Real;
               SP_PumpSpeed : Real;
            END_STRUCT;
            ProWater : Struct
               Sp_DoseQty : Real;
               SP_PumpSpeed : Real;
            END_STRUCT;
            Homomixer : Struct
               Sp_DoseQty : Real;
               SP_PumpSpeed : Real;
            END_STRUCT;
         END_STRUCT;
         "T-21" : Struct
            HW : Struct
               Sp_Flush_to_BlendQty : Real;
               Sp_Flush_to_DrainQty : Real;
               Sp_DrainTime : DInt;
               SP_PumpSpeed : Real;
            END_STRUCT;
            ChiliAwetan_1 : Struct
               Sp_DoseQty : Real;
               SP_PumpSpeed : Real;
            END_STRUCT;
            ChiliAwetan_2 : Struct
               Sp_DoseQty : Real;
               SP_PumpSpeed : Real;
            END_STRUCT;
            ChiliAwetan_3 : Struct
               Sp_DoseQty : Real;
               SP_PumpSpeed : Real;
            END_STRUCT;
            Tomato : Struct
               Sp_DoseQty : Real;
               SP_PumpSpeed : Real;
            END_STRUCT;
            ChiliFresh_1 : Struct
               Sp_DoseQty : Real;
               SP_PumpSpeed : Real;
            END_STRUCT;
            ChiliFresh_2 : Struct
               Sp_DoseQty : Real;
               SP_PumpSpeed : Real;
            END_STRUCT;
            ChiliFresh_3 : Struct
               Sp_DoseQty : Real;
               SP_PumpSpeed : Real;
            END_STRUCT;
            Garlic : Struct
               Sp_DoseQty : Real;
               SP_PumpSpeed : Real;
            END_STRUCT;
            Vinegar : Struct
               Sp_DoseQty : Real;
               SP_PumpSpeed : Real;
            END_STRUCT;
            Sugar : Struct
               Sp_DoseQty : Real;
               SP_PumpSpeed : Real;
            END_STRUCT;
            Salt : Struct
               Sp_DoseQty : Real;
               SP_PumpSpeed : Real;
            END_STRUCT;
            ProWater : Struct
               Sp_DoseQty : Real;
               SP_PumpSpeed : Real;
            END_STRUCT;
            Homomixer : Struct
               Sp_DoseQty : Real;
               SP_PumpSpeed : Real;
            END_STRUCT;
         END_STRUCT;
         "T-30" : Struct
            HW : Struct
               Sp_Flush_to_BlendQty : Real;
               Sp_Flush_to_DrainQty : Real;
               Sp_DrainTime : DInt;
               SP_PumpSpeed : Real;
            END_STRUCT;
            ChiliAwetan_1 : Struct
               Sp_DoseQty : Real;
               SP_PumpSpeed : Real;
            END_STRUCT;
            ChiliAwetan_2 : Struct
               Sp_DoseQty : Real;
               SP_PumpSpeed : Real;
            END_STRUCT;
            ChiliAwetan_3 : Struct
               Sp_DoseQty : Real;
               SP_PumpSpeed : Real;
            END_STRUCT;
            Tomato : Struct
               Sp_DoseQty : Real;
               SP_PumpSpeed : Real;
            END_STRUCT;
            ChiliFresh_1 : Struct
               Sp_DoseQty : Real;
               SP_PumpSpeed : Real;
            END_STRUCT;
            ChiliFresh_2 : Struct
               Sp_DoseQty : Real;
               SP_PumpSpeed : Real;
            END_STRUCT;
            ChiliFresh_3 : Struct
               Sp_DoseQty : Real;
               SP_PumpSpeed : Real;
            END_STRUCT;
            Garlic : Struct
               Sp_DoseQty : Real;
               SP_PumpSpeed : Real;
            END_STRUCT;
            Vinegar : Struct
               Sp_DoseQty : Real;
               SP_PumpSpeed : Real;
            END_STRUCT;
            Sugar : Struct
               Sp_DoseQty : Real;
               SP_PumpSpeed : Real;
            END_STRUCT;
            Salt : Struct
               Sp_DoseQty : Real;
               SP_PumpSpeed : Real;
            END_STRUCT;
            ProWater : Struct
               Sp_DoseQty : Real;
               SP_PumpSpeed : Real;
            END_STRUCT;
            Homomixer : Struct
               Sp_DoseQty : Real;
               SP_PumpSpeed : Real;
            END_STRUCT;
         END_STRUCT;
         "T-31" : Struct
            HW : Struct
               Sp_Flush_to_BlendQty : Real;
               Sp_Flush_to_DrainQty : Real;
               Sp_DrainTime : DInt;
               SP_PumpSpeed : Real;
            END_STRUCT;
            ChiliAwetan_1 : Struct
               Sp_DoseQty : Real;
               SP_PumpSpeed : Real;
            END_STRUCT;
            ChiliAwetan_2 : Struct
               Sp_DoseQty : Real;
               SP_PumpSpeed : Real;
            END_STRUCT;
            ChiliAwetan_3 : Struct
               Sp_DoseQty : Real;
               SP_PumpSpeed : Real;
            END_STRUCT;
            Tomato : Struct
               Sp_DoseQty : Real;
               SP_PumpSpeed : Real;
            END_STRUCT;
            ChiliFresh_1 : Struct
               Sp_DoseQty : Real;
               SP_PumpSpeed : Real;
            END_STRUCT;
            ChiliFresh_2 : Struct
               Sp_DoseQty : Real;
               SP_PumpSpeed : Real;
            END_STRUCT;
            ChiliFresh_3 : Struct
               Sp_DoseQty : Real;
               SP_PumpSpeed : Real;
            END_STRUCT;
            Garlic : Struct
               Sp_DoseQty : Real;
               SP_PumpSpeed : Real;
            END_STRUCT;
            Vinegar : Struct
               Sp_DoseQty : Real;
               SP_PumpSpeed : Real;
            END_STRUCT;
            Sugar : Struct
               Sp_DoseQty : Real;
               SP_PumpSpeed : Real;
            END_STRUCT;
            Salt : Struct
               Sp_DoseQty : Real;
               SP_PumpSpeed : Real;
            END_STRUCT;
            ProWater : Struct
               Sp_DoseQty : Real;
               SP_PumpSpeed : Real;
            END_STRUCT;
            Homomixer : Struct
               Sp_DoseQty : Real;
               SP_PumpSpeed : Real;
            END_STRUCT;
         END_STRUCT;
         "T-40" : Struct
            HW : Struct
               Sp_Flush_to_BlendQty : Real;
               Sp_Flush_to_DrainQty : Real;
               Sp_DrainTime : DInt;
               SP_PumpSpeed : Real;
            END_STRUCT;
            ChiliAwetan_1 : Struct
               Sp_DoseQty : Real;
               SP_PumpSpeed : Real;
            END_STRUCT;
            ChiliAwetan_2 : Struct
               Sp_DoseQty : Real;
               SP_PumpSpeed : Real;
            END_STRUCT;
            ChiliAwetan_3 : Struct
               Sp_DoseQty : Real;
               SP_PumpSpeed : Real;
            END_STRUCT;
            Tomato : Struct
               Sp_DoseQty : Real;
               SP_PumpSpeed : Real;
            END_STRUCT;
            ChiliFresh_1 : Struct
               Sp_DoseQty : Real;
               SP_PumpSpeed : Real;
            END_STRUCT;
            ChiliFresh_2 : Struct
               Sp_DoseQty : Real;
               SP_PumpSpeed : Real;
            END_STRUCT;
            ChiliFresh_3 : Struct
               Sp_DoseQty : Real;
               SP_PumpSpeed : Real;
            END_STRUCT;
            Garlic : Struct
               Sp_DoseQty : Real;
               SP_PumpSpeed : Real;
            END_STRUCT;
            Vinegar : Struct
               Sp_DoseQty : Real;
               SP_PumpSpeed : Real;
            END_STRUCT;
            Sugar : Struct
               Sp_DoseQty : Real;
               SP_PumpSpeed : Real;
            END_STRUCT;
            Salt : Struct
               Sp_DoseQty : Real;
               SP_PumpSpeed : Real;
            END_STRUCT;
            ProWater : Struct
               Sp_DoseQty : Real;
               SP_PumpSpeed : Real;
            END_STRUCT;
            Homomixer : Struct
               Sp_DoseQty : Real;
               SP_PumpSpeed : Real;
            END_STRUCT;
         END_STRUCT;
         "T-41" : Struct
            HW : Struct
               Sp_Flush_to_BlendQty : Real;
               Sp_Flush_to_DrainQty : Real;
               Sp_DrainTime : DInt;
               SP_PumpSpeed : Real;
            END_STRUCT;
            ChiliAwetan_1 : Struct
               Sp_DoseQty : Real;
               SP_PumpSpeed : Real;
            END_STRUCT;
            ChiliAwetan_2 : Struct
               Sp_DoseQty : Real;
               SP_PumpSpeed : Real;
            END_STRUCT;
            ChiliAwetan_3 : Struct
               Sp_DoseQty : Real;
               SP_PumpSpeed : Real;
            END_STRUCT;
            Tomato : Struct
               Sp_DoseQty : Real;
               SP_PumpSpeed : Real;
            END_STRUCT;
            ChiliFresh_1 : Struct
               Sp_DoseQty : Real;
               SP_PumpSpeed : Real;
            END_STRUCT;
            ChiliFresh_2 : Struct
               Sp_DoseQty : Real;
               SP_PumpSpeed : Real;
            END_STRUCT;
            ChiliFresh_3 : Struct
               Sp_DoseQty : Real;
               SP_PumpSpeed : Real;
            END_STRUCT;
            Garlic : Struct
               Sp_DoseQty : Real;
               SP_PumpSpeed : Real;
            END_STRUCT;
            Vinegar : Struct
               Sp_DoseQty : Real;
               SP_PumpSpeed : Real;
            END_STRUCT;
            Sugar : Struct
               Sp_DoseQty : Real;
               SP_PumpSpeed : Real;
            END_STRUCT;
            Salt : Struct
               Sp_DoseQty : Real;
               SP_PumpSpeed : Real;
            END_STRUCT;
            ProWater : Struct
               Sp_DoseQty : Real;
               SP_PumpSpeed : Real;
            END_STRUCT;
            Homomixer : Struct
               Sp_DoseQty : Real;
               SP_PumpSpeed : Real;
            END_STRUCT;
         END_STRUCT;
      END_STRUCT;
   END_VAR
   VAR
      ProdReq_Header_1 : Bool;
      ProdReq_Header_2 : Bool;
      freeBool_3 : Bool;
      freeBool_4 : Bool;
      freeBool_5 : Bool;
      freeBool_6 : Bool;
      freeBool_7 : Bool;
      freeBool_8 : Bool;
      freeBool_9 : Bool;
      freeBool_10 : Bool;
      freeBool_11 : Bool;
      freeBool_12 : Bool;
      freeBool_13 : Bool;
      freeBool_14 : Bool;
      freeBool_15 : Bool;
      freeBool_16 : Bool;
      freeReal_1 : Real;
      freeReal_2 : Real;
      freeReal_3 : Real;
      freeReal_4 : Real;
      freeReal_5 : Real;
      freeReal_6 : Real;
      freeReal_7 : Real;
      freeReal_8 : Real;
      freeReal_9 : Real;
      freeReal_10 : Real;
      freeReal_11 : Real;
      freeReal_12 : Real;
      freeReal_13 : Real;
      freeReal_14 : Real;
      freeReal_15 : Real;
      freeReal_16 : Real;
   END_VAR
BEGIN
END_DATA_BLOCK

